  MoveC 5250 to (-74.2, -30.87, -8) mm, rotated rx 180 ry 0 rz 90 deg; joints [72.057, -18.552, 88.853, 0, 19.699, 72.057] to (-74.66, -32.55, -8) mm, rotated rx -180 ry 0 rz 90 deg; joints [71.996, -18.551, 88.847, 0, 19.704, 71.996]
  MoveL 5251 to (-74.66, -70.65, -8) mm, rotated rx 180 ry 0 rz 90 deg; joints [70.74, -18.352, 87.987, 0, 20.365, 70.74]
  MoveC 5252 to (-73.67, -73.03, -8) mm, rotated rx 180 ry 0 rz 90 deg; joints [70.673, -18.323, 87.865, 0, 20.458, 70.673] to (-71.29, -74.01, -8) mm, rotated rx 180 ry 0 rz 90 deg; joints [70.668, -18.28, 87.682, 0, 20.598, 70.668]
  MoveC 5253 to (-53.37, -73.92, -8) mm, rotated rx 180 ry 0 rz 90 deg; joints [70.874, -17.988, 86.471, 0, 21.517, 70.874] to (-35.45, -73.74, -8) mm, rotated rx 180 ry 0 rz 90 deg; joints [71.079, -17.682, 85.244, 0, 22.437, 71.079]
  MoveC 5254 to (-33.46, -73.06, -8) mm, rotated rx 180 ry 0 rz 90 deg; joints [71.123, -17.651, 85.123, 0, 22.528, 71.123] to (-32.27, -71.32, -8) mm, rotated rx 180 ry 0 rz 90 deg; joints [71.192, -17.64, 85.081, 0, 22.559, 71.192]
  MoveC 5255 to (-31.64, -69.07, -8) mm, rotated rx 180 ry 0 rz 90 deg; joints [71.27, -17.643, 85.091, 0, 22.552, 71.27] to (-31.06, -66.81, -8) mm, rotated rx 180 ry 0 rz 90 deg; joints [71.349, -17.646, 85.103, 0, 22.542, 71.349]
  MoveL 5256 to (-30.8, -65.76, -8) mm, rotated rx 180 ry 0 rz 90 deg; joints [71.386, -17.647, 85.11, 0, 22.537, 71.386]
  MoveC 5257 to (-25.24, -44.49, -8) mm, rotated rx -180 ry 0 rz 90 deg; joints [72.129, -17.673, 85.211, 0, 22.462, 72.129] to (-19.72, -23.22, -8) mm, rotated rx -180 ry 0 rz 90 deg; joints [72.873, -17.694, 85.294, 0, 22.401, 72.873]
  MoveC 5258 to (-19.64, -22.75, -8) mm, rotated rx -180 ry 0 rz 90 deg; joints [72.889, -17.695, 85.299, 0, 22.397, 72.889] to (-19.7, -22.27, -8) mm, rotated rx 180 ry 0 rz 90 deg; joints [72.904, -17.699, 85.313, 0, 22.386, 72.904]
  MoveC 5259 to (-20.47, -20.62, -8) mm, rotated rx 180 ry 0 rz 90 deg; joints [72.949, -17.721, 85.402, 0, 22.319, 72.949] to (-21.84, -19.43, -8) mm, rotated rx -180 ry 0 rz 90 deg; joints [72.975, -17.752, 85.523, 0, 22.229, 72.975]
  MoveL 5260 to (-22.21, -19.24, -8) mm, rotated rx -180 ry 0 rz 90 deg; joints [72.977, -17.76, 85.553, 0, 22.206, 72.977]
  MoveC 5261 to (-22.95, -19.01, -8) mm, rotated rx -180 ry 0 rz 90 deg; joints [72.977, -17.774, 85.609, 0, 22.164, 72.977] to (-23.72, -19.03, -8) mm, rotated rx 180 ry 0 rz 90 deg; joints [72.969, -17.787, 85.663, 0, 22.124, 72.969]
  MoveL 5262 to (-32.69, -20.92, -8) mm, rotated rx -180 ry 0 rz 90 deg; joints [72.817, -17.932, 86.244, 0, 21.687, 72.817]
  MoveL 5263 to (-47.78, -24.13, -8) mm, rotated rx 180 ry 0 rz 90 deg; joints [72.558, -18.168, 87.212, 0, 20.956, 72.558]
  MoveL 5264 to (-46.21, -31.51, -8) mm, rotated rx 180 ry 0 rz 90 deg; joints [72.332, -18.103, 86.945, 0, 21.158, 72.332]
  MoveL 5265 to (-46.21, -31.51, -5) mm, rotated rx 180 ry 0 rz 90 deg; joints [72.332, -18.259, 87.047, 0, 21.212, 72.332]
  Establecer velocidad (1000.0 mm/s)
  MoveL 5266 to (-46.21, -31.51, 10) mm, rotated rx 180 ry 0 rz 90 deg; joints [72.332, -19.034, 87.547, 0, 21.486, 72.332]
  Establecer velocidad (66.7 mm/s)
  MoveL 5267 to (15.53, -65.29, 10) mm, rotated rx -180 ry 0 rz 90 deg; joints [71.889, -17.693, 82.447, 0, 25.246, 71.889]
  MoveL 5268 to (15.53, -65.29, -4.75) mm, rotated rx -180 ry 0 rz 90 deg; joints [71.889, -16.947, 81.953, 0, 24.994, 71.889]
  MoveL 5269 to (15.38, -66.79, -5.16) mm, rotated rx 180 ry 0 rz 90 deg; joints [71.84, -16.919, 81.915, 0, 25.005, 71.84]
  MoveL 5270 to (15.6, -68.3, -5.56) mm, rotated rx -180 ry 0 rz 90 deg; joints [71.795, -16.885, 81.85, 0, 25.035, 71.795]
  MoveL 5271 to (16.14, -69.72, -5.97) mm, rotated rx 180 ry 0 rz 90 deg; joints [71.756, -16.844, 81.763, 0, 25.081, 71.756]
  MoveL 5272 to (16.98, -70.99, -6.38) mm, rotated rx -180 ry 0 rz 90 deg; joints [71.725, -16.798, 81.659, 0, 25.14, 71.725]
  MoveL 5273 to (18.08, -72.03, -6.78) mm, rotated rx -180 ry 0 rz 90 deg; joints [71.704, -16.749, 81.54, 0, 25.209, 71.704]
  MoveL 5274 to (19.39, -72.81, -7.19) mm, rotated rx -180 ry 0 rz 90 deg; joints [71.693, -16.697, 81.413, 0, 25.284, 71.693]
  MoveL 5275 to (20.83, -73.28, -7.59) mm, rotated rx 180 ry 0 rz 90 deg; joints [71.693, -16.644, 81.283, 0, 25.361, 71.693]
  MoveL 5276 to (22.34, -73.39, -8) mm, rotated rx -180 ry 0 rz 90 deg; joints [71.705, -16.592, 81.157, 0, 25.435, 71.705]
  MoveC 5277 to (34.58, -73.11, -8) mm, rotated rx 180 ry 0 rz 90 deg; joints [71.839, -16.343, 80.27, 0, 26.073, 71.839] to (46.81, -72.79, -8) mm, rotated rx -180 ry 0 rz 90 deg; joints [71.972, -16.086, 79.374, 0, 26.712, 71.972]
  MoveC 5278 to (49.35, -69.79, -8) mm, rotated rx -180 ry 0 rz 90 deg; joints [72.09, -16.053, 79.258, 0, 26.795, 72.09] to (49.49, -65.86, -8) mm, rotated rx -180 ry 0 rz 90 deg; joints [72.213, -16.077, 79.342, 0, 26.735, 72.213]
  MoveL 5279 to (48.8, -64.98, -8) mm, rotated rx 180 ry 0 rz 90 deg; joints [72.233, -16.098, 79.414, 0, 26.684, 72.233]
  MoveL 5280 to (42.36, -57.33, -8) mm, rotated rx 180 ry 0 rz 90 deg; joints [72.406, -16.286, 80.072, 0, 26.215, 72.406]
  MoveL 5281 to (25.46, -37.43, -8) mm, rotated rx -180 ry 0 rz 90 deg; joints [72.864, -16.761, 81.765, 0, 24.996, 72.864]
  MoveL 5282 to (25.29, -37.24, -8) mm, rotated rx -180 ry 0 rz 90 deg; joints [72.868, -16.765, 81.782, 0, 24.984, 72.868]
  MoveC 5283 to (24.85, -36.79, -8) mm, rotated rx -180 ry 0 rz 90 deg; joints [72.878, -16.777, 81.824, 0, 24.953, 72.878] to (24.37, -36.38, -8) mm, rotated rx 180 ry 0 rz 90 deg; joints [72.886, -16.789, 81.867, 0, 24.921, 72.886]
  MoveL 5284 to (12.74, -27.01, -8) mm, rotated rx -180 ry 0 rz 90 deg; joints [73.07, -17.073, 82.914, 0, 24.159, 73.07]
  MoveL 5285 to (12.32, -26.68, -8) mm, rotated rx -180 ry 0 rz 90 deg; joints [73.077, -17.083, 82.951, 0, 24.132, 73.077]
  MoveC 5286 to (9.55, -26.29, -8) mm, rotated rx -180 ry 0 rz 90 deg; joints [73.062, -17.138, 83.158, 0, 23.98, 73.062] to (7.11, -27.65, -8) mm, rotated rx -180 ry 0 rz 90 deg; joints [72.995, -17.177, 83.303, 0, 23.874, 72.995]
  MoveC 5287 to (6.83, -28.04, -8) mm, rotated rx -180 ry 0 rz 90 deg; joints [72.98, -17.18, 83.314, 0, 23.866, 72.98] to (6.65, -28.48, -8) mm, rotated rx -180 ry 0 rz 90 deg; joints [72.964, -17.181, 83.317, 0, 23.864, 72.964]
  MoveL 5288 to (-4.13, -68.7, -8) mm, rotated rx 180 ry 0 rz 90 deg; joints [71.576, -17.141, 83.169, 0, 23.972, 71.576]
  MoveL 5289 to (-4.25, -69.18, -8) mm, rotated rx 180 ry 0 rz 90 deg; joints [71.56, -17.141, 83.167, 0, 23.974, 71.56]
  MoveC 5290 to (-3.94, -71.7, -8) mm, rotated rx -180 ry 0 rz 90 deg; joints [71.484, -17.119, 83.085, 0, 24.034, 71.484] to (-2.08, -73.44, -8) mm, rotated rx -180 ry 0 rz 90 deg; joints [71.448, -17.072, 82.911, 0, 24.161, 71.448]
  MoveL 5291 to (-1.42, -73.69, -8) mm, rotated rx -180 ry 0 rz 90 deg; joints [71.447, -17.058, 82.858, 0, 24.2, 71.447]
  MoveL 5292 to (-0.47, -73.77, -8) mm, rotated rx 180 ry 0 rz 90 deg; joints [71.455, -17.039, 82.789, 0, 24.25, 71.455]
  MoveC 5293 to (10.93, -73.6, -8) mm, rotated rx -180 ry 0 rz 90 deg; joints [71.58, -16.819, 81.977, 0, 24.842, 71.58] to (22.34, -73.39, -8) mm, rotated rx -180 ry 0 rz 90 deg; joints [71.705, -16.592, 81.157, 0, 25.435, 71.705]
  MoveL 5294 to (22.19, -65.84, -8) mm, rotated rx -180 ry 0 rz 90 deg; joints [71.939, -16.645, 81.348, 0, 25.297, 71.939]
  MoveL 5295 to (22.19, -65.84, -5) mm, rotated rx -180 ry 0 rz 90 deg; joints [71.939, -16.797, 81.45, 0, 25.347, 71.939]
  Establecer velocidad (1000.0 mm/s)
  MoveL 5296 to (22.19, -65.84, 10) mm, rotated rx 180 ry 0 rz 90 deg; joints [71.939, -17.555, 81.953, 0, 25.602, 71.939]
  Establecer velocidad (66.7 mm/s)
  MoveL 5297 to (63.14, -31.68, 10) mm, rotated rx -180 ry 0 rz 90 deg; joints [73.4, -16.913, 79.72, 0, 27.194, 73.4]
  MoveL 5298 to (63.14, -31.68, -4.75) mm, rotated rx -180 ry 0 rz 90 deg; joints [73.4, -16.174, 79.223, 0, 26.951, 73.4]
  MoveL 5299 to (64.65, -31.87, -5.16) mm, rotated rx 180 ry 0 rz 90 deg; joints [73.409, -16.119, 79.092, 0, 27.027, 73.409]
  MoveL 5300 to (66.16, -31.68, -5.56) mm, rotated rx 180 ry 0 rz 90 deg; joints [73.428, -16.067, 78.969, 0, 27.098, 73.428]
  MoveL 5301 to (67.59, -31.17, -5.97) mm, rotated rx 180 ry 0 rz 90 deg; joints [73.457, -16.019, 78.859, 0, 27.16, 73.457]
  MoveL 5302 to (68.87, -30.36, -6.38) mm, rotated rx 180 ry 0 rz 90 deg; joints [73.494, -15.975, 78.766, 0, 27.209, 73.494]
  MoveL 5303 to (69.94, -29.28, -6.78) mm, rotated rx -180 ry 0 rz 90 deg; joints [73.537, -15.938, 78.696, 0, 27.243, 73.537]
  MoveL 5304 to (70.74, -27.99, -7.19) mm, rotated rx 180 ry 0 rz 90 deg; joints [73.584, -15.909, 78.65, 0, 27.259, 73.584]
  MoveL 5305 to (71.24, -26.55, -7.59) mm, rotated rx 180 ry 0 rz 90 deg; joints [73.633, -15.887, 78.63, 0, 27.256, 73.633]
  MoveL 5306 to (71.38, -25.04, -8) mm, rotated rx 180 ry 0 rz 90 deg; joints [73.681, -15.873, 78.639, 0, 27.234, 73.681]
  MoveL 5307 to (71.38, -16.01, -8) mm, rotated rx 180 ry 0 rz 90 deg; joints [73.961, -15.931, 78.837, 0, 27.094, 73.961]
  MoveC 5308 to (69.58, -13.38, -8) mm, rotated rx 180 ry 0 rz 90 deg; joints [74.027, -15.987, 79.03, 0, 26.957, 74.027] to (66.81, -11.79, -8) mm, rotated rx -180 ry 0 rz 90 deg; joints [74.052, -16.057, 79.273, 0, 26.784, 74.052]
  MoveC 5309 to (65.71, -11.6, -8) mm, rotated rx 180 ry 0 rz 90 deg; joints [74.047, -16.082, 79.36, 0, 26.723, 74.047] to (64.59, -11.73, -8) mm, rotated rx -180 ry 0 rz 90 deg; joints [74.034, -16.106, 79.44, 0, 26.665, 74.034]
  MoveL 5310 to (56.12, -23.22, -8) mm, rotated rx 180 ry 0 rz 90 deg; joints [73.599, -16.216, 79.824, 0, 26.392, 73.599]
  MoveL 5311 to (55.62, -23.94, -8) mm, rotated rx -180 ry 0 rz 90 deg; joints [73.572, -16.222, 79.846, 0, 26.376, 73.572]
  MoveC 5312 to (55.02, -26.08, -8) mm, rotated rx -180 ry 0 rz 90 deg; joints [73.5, -16.221, 79.844, 0, 26.378, 73.5] to (55.87, -28.13, -8) mm, rotated rx 180 ry 0 rz 90 deg; joints [73.444, -16.19, 79.735, 0, 26.456, 73.444]
  MoveL 5313 to (64.98, -38.32, -8) mm, rotated rx -180 ry 0 rz 90 deg; joints [73.212, -15.927, 78.824, 0, 27.103, 73.212]
  MoveC 5314 to (66.47, -38.38, -8) mm, rotated rx 180 ry 0 rz 90 deg; joints [73.224, -15.894, 78.711, 0, 27.183, 73.224] to (67.89, -37.93, -8) mm, rotated rx -180 ry 0 rz 90 deg; joints [73.251, -15.866, 78.614, 0, 27.251, 73.251]
  MoveL 5315 to (68.22, -37.76, -8) mm, rotated rx 180 ry 0 rz 90 deg; joints [73.259, -15.859, 78.593, 0, 27.266, 73.259]
  MoveC 5316 to (70.16, -36.22, -8) mm, rotated rx -180 ry 0 rz 90 deg; joints [73.325, -15.827, 78.482, 0, 27.345, 73.325] to (71.38, -34.07, -8) mm, rotated rx -180 ry 0 rz 90 deg; joints [73.402, -15.814, 78.437, 0, 27.376, 73.402]
  MoveL 5317 to (71.38, -25.04, -8) mm, rotated rx 180 ry 0 rz 90 deg; joints [73.681, -15.873, 78.639, 0, 27.234, 73.681]
  MoveL 5318 to (63.83, -25.04, -8) mm, rotated rx 180 ry 0 rz 90 deg; joints [73.613, -16.038, 79.208, 0, 26.831, 73.613]
  MoveL 5319 to (63.83, -25.48, -8) mm, rotated rx -180 ry 0 rz 90 deg; joints [73.599, -16.036, 79.198, 0, 26.838, 73.599]
  MoveL 5320 to (63.83, -25.48, -5) mm, rotated rx 180 ry 0 rz 90 deg; joints [73.599, -16.186, 79.301, 0, 26.886, 73.599]
  Establecer velocidad (1000.0 mm/s)
  MoveL 5321 to (63.83, -25.48, 10) mm, rotated rx -180 ry 0 rz 90 deg; joints [73.599, -16.939, 79.806, 0, 27.133, 73.599]
  Establecer velocidad (66.7 mm/s)
  MoveL 5322 to (31.82, 9.28, 10) mm, rotated rx -180 ry 0 rz 90 deg; joints [74.404, -17.82, 82.904, 0, 24.916, 74.404]
  MoveL 5323 to (31.82, 9.28, -4.75) mm, rotated rx 180 ry 0 rz 90 deg; joints [74.404, -17.072, 82.41, 0, 24.662, 74.404]
  MoveL 5324 to (32.94, 8.26, -5.16) mm, rotated rx 180 ry 0 rz 90 deg; joints [74.381, -17.024, 82.294, 0, 24.729, 74.381]
  MoveL 5325 to (34.28, 7.54, -5.56) mm, rotated rx 180 ry 0 rz 90 deg; joints [74.37, -16.972, 82.168, 0, 24.804, 74.37]
  MoveL 5326 to (35.74, 7.13, -5.97) mm, rotated rx -180 ry 0 rz 90 deg; joints [74.37, -16.92, 82.039, 0, 24.881, 74.37]
  MoveL 5327 to (37.26, 7.06, -6.38) mm, rotated rx 180 ry 0 rz 90 deg; joints [74.382, -16.869, 81.913, 0, 24.955, 74.382]
  MoveL 5328 to (38.76, 7.32, -6.78) mm, rotated rx 180 ry 0 rz 90 deg; joints [74.403, -16.819, 81.795, 0, 25.024, 74.403]
  MoveL 5329 to (40.15, 7.91, -7.19) mm, rotated rx 180 ry 0 rz 90 deg; joints [74.434, -16.774, 81.691, 0, 25.083, 74.434]
  MoveL 5330 to (41.39, 8.8, -7.59) mm, rotated rx 180 ry 0 rz 90 deg; joints [74.473, -16.733, 81.605, 0, 25.129, 74.473]
  MoveL 5331 to (42.37, 9.95, -8) mm, rotated rx 180 ry 0 rz 90 deg; joints [74.519, -16.699, 81.542, 0, 25.157, 74.519]
  MoveL 5332 to (51.07, 22.27, -8) mm, rotated rx 180 ry 0 rz 90 deg; joints [74.985, -16.59, 81.149, 0, 25.441, 74.985]
  MoveC 5333 to (50.81, 26.19, -8) mm, rotated rx 180 ry 0 rz 90 deg; joints [75.107, -16.617, 81.245, 0, 25.371, 75.107] to (48.1, 29.04, -8) mm, rotated rx 180 ry 0 rz 90 deg; joints [75.175, -16.688, 81.501, 0, 25.187, 75.175]
  MoveC 5334 to (29.5, 28.81, -8) mm, rotated rx -180 ry 0 rz 90 deg; joints [75.009, -17.057, 82.856, 0, 24.201, 75.009] to (10.9, 28.45, -8) mm, rotated rx 180 ry 0 rz 90 deg; joints [74.836, -17.41, 84.188, 0, 23.222, 74.836]
  MoveC 5335 to (8.09, 27.12, -8) mm, rotated rx 180 ry 0 rz 90 deg; joints [74.768, -17.455, 84.362, 0, 23.093, 74.768] to (7.1, 24.17, -8) mm, rotated rx 180 ry 0 rz 90 deg; joints [74.663, -17.459, 84.375, 0, 23.084, 74.663]
  MoveC 5336 to (7.15, 23.93, -8) mm, rotated rx 180 ry 0 rz 90 deg; joints [74.656, -17.457, 84.367, 0, 23.089, 74.656] to (7.21, 23.7, -8) mm, rotated rx -180 ry 0 rz 90 deg; joints [74.649, -17.454, 84.358, 0, 23.096, 74.649]
  MoveL 5337 to (11.88, 10.9, -8) mm, rotated rx -180 ry 0 rz 90 deg; joints [74.277, -17.301, 83.771, 0, 23.53, 74.277]
  MoveL 5338 to (12.28, 9.83, -8) mm, rotated rx -180 ry 0 rz 90 deg; joints [74.246, -17.288, 83.721, 0, 23.567, 74.246]
  MoveC 5339 to (12.77, 8.93, -8) mm, rotated rx 180 ry 0 rz 90 deg; joints [74.221, -17.274, 83.668, 0, 23.606, 74.221] to (13.49, 8.19, -8) mm, rotated rx -180 ry 0 rz 90 deg; joints [74.204, -17.256, 83.601, 0, 23.655, 74.204]
  MoveL 5340 to (27.96, -2.86, -8) mm, rotated rx -180 ry 0 rz 90 deg; joints [73.982, -16.915, 82.331, 0, 24.585, 73.982]
  MoveL 5341 to (28.9, -3.52, -8) mm, rotated rx 180 ry 0 rz 90 deg; joints [73.97, -16.893, 82.248, 0, 24.645, 73.97]
  MoveC 5342 to (31.47, -3.69, -8) mm, rotated rx -180 ry 0 rz 90 deg; joints [73.988, -16.841, 82.058, 0, 24.783, 73.988] to (33.68, -2.37, -8) mm, rotated rx -180 ry 0 rz 90 deg; joints [74.05, -16.804, 81.924, 0, 24.88, 74.05]
  MoveL 5343 to (42.37, 9.95, -8) mm, rotated rx 180 ry 0 rz 90 deg; joints [74.519, -16.699, 81.542, 0, 25.157, 74.519]
  MoveL 5344 to (36.21, 14.3, -8) mm, rotated rx -180 ry 0 rz 90 deg; joints [74.603, -16.847, 82.081, 0, 24.766, 74.603]
  MoveL 5345 to (36.21, 14.3, -5) mm, rotated rx 180 ry 0 rz 90 deg; joints [74.603, -17, 82.183, 0, 24.816, 74.603]
  Establecer velocidad (1000.0 mm/s)
  MoveL 5346 to (36.21, 14.3, 10) mm, rotated rx 180 ry 0 rz 90 deg; joints [74.603, -17.76, 82.686, 0, 25.074, 74.603]
  Establecer velocidad (66.7 mm/s)
  MoveL 5347 to (28.17, 64.78, 10) mm, rotated rx 180 ry 0 rz 90 deg; joints [76.16, -18.179, 84.225, 0, 23.954, 76.16]
  MoveL 5348 to (28.17, 64.78, -4.75) mm, rotated rx 180 ry 0 rz 90 deg; joints [76.16, -17.427, 83.732, 0, 23.695, 76.16]
  MoveL 5349 to (28.39, 66.28, -5.16) mm, rotated rx -180 ry 0 rz 90 deg; joints [76.21, -17.41, 83.729, 0, 23.68, 76.21]
  MoveL 5350 to (28.24, 67.79, -5.56) mm, rotated rx 180 ry 0 rz 90 deg; joints [76.258, -17.399, 83.753, 0, 23.645, 76.258]
  MoveL 5351 to (27.76, 69.23, -5.97) mm, rotated rx 180 ry 0 rz 90 deg; joints [76.302, -17.394, 83.8, 0, 23.594, 76.302]
  MoveL 5352 to (26.97, 70.53, -6.38) mm, rotated rx 180 ry 0 rz 90 deg; joints [76.338, -17.394, 83.865, 0, 23.529, 76.338]
  MoveL 5353 to (25.91, 71.63, -6.78) mm, rotated rx -180 ry 0 rz 90 deg; joints [76.365, -17.398, 83.947, 0, 23.451, 76.365]
  MoveL 5354 to (24.64, 72.46, -7.19) mm, rotated rx 180 ry 0 rz 90 deg; joints [76.382, -17.405, 84.039, 0, 23.366, 76.382]
  MoveL 5355 to (23.22, 72.99, -7.59) mm, rotated rx -180 ry 0 rz 90 deg; joints [76.388, -17.414, 84.137, 0, 23.277, 76.388]
  MoveL 5356 to (21.71, 73.16, -8) mm, rotated rx -180 ry 0 rz 90 deg; joints [76.382, -17.422, 84.235, 0, 23.187, 76.382]
  MoveL 5357 to (16.58, 73.28, -8) mm, rotated rx -180 ry 0 rz 90 deg; joints [76.345, -17.518, 84.605, 0, 22.913, 76.345]
  MoveL 5358 to (-23.22, 73.93, -8) mm, rotated rx 180 ry 0 rz 90 deg; joints [76.043, -18.217, 87.419, 0, 20.798, 76.043]
  MoveL 5359 to (-24.65, 73.95, -8) mm, rotated rx 180 ry 0 rz 90 deg; joints [76.031, -18.241, 87.519, 0, 20.722, 76.031]
  MoveC 5360 to (-27.16, 70.81, -8) mm, rotated rx -180 ry 0 rz 90 deg; joints [75.905, -18.269, 87.638, 0, 20.632, 75.905] to (-26.78, 66.82, -8) mm, rotated rx 180 ry 0 rz 90 deg; joints [75.774, -18.247, 87.542, 0, 20.705, 75.774]
  MoveL 5361 to (-9, 55.49, -8) mm, rotated rx 180 ry 0 rz 90 deg; joints [75.549, -17.897, 86.102, 0, 21.795, 75.549]
  MoveL 5362 to (-8.91, 55.44, -8) mm, rotated rx -180 ry 0 rz 90 deg; joints [75.548, -17.895, 86.094, 0, 21.801, 75.548]
  MoveL 5363 to (-8.41, 55.2, -8) mm, rotated rx -180 ry 0 rz 90 deg; joints [75.544, -17.885, 86.055, 0, 21.83, 75.544]
  MoveL 5364 to (-8.28, 55.16, -8) mm, rotated rx -180 ry 0 rz 90 deg; joints [75.544, -17.883, 86.046, 0, 21.837, 75.544]
  MoveC 5365 to (-7.7, 55.1, -8) mm, rotated rx 180 ry 0 rz 90 deg; joints [75.547, -17.872, 86.004, 0, 21.869, 75.547] to (-7.11, 55.11, -8) mm, rotated rx 180 ry 0 rz 90 deg; joints [75.552, -17.862, 85.962, 0, 21.9, 75.552]
  MoveC 5366 to (9.95, 56.35, -8) mm, rotated rx 180 ry 0 rz 90 deg; joints [75.737, -17.562, 84.778, 0, 22.785, 75.737] to (27.01, 57.72, -8) mm, rotated rx 180 ry 0 rz 90 deg; joints [75.922, -17.25, 83.579, 0, 23.671, 75.922]
  MoveC 5367 to (45.69, 59.55, -8) mm, rotated rx -180 ry 0 rz 90 deg; joints [76.131, -16.894, 82.252, 0, 24.642, 76.131] to (64.31, 62.01, -8) mm, rotated rx 180 ry 0 rz 90 deg; joints [76.355, -16.526, 80.92, 0, 25.606, 76.355]
  MoveC 5368 to (66.34, 62.34, -8) mm, rotated rx 180 ry 0 rz 90 deg; joints [76.381, -16.485, 80.774, 0, 25.711, 76.381] to (68.36, 62.74, -8) mm, rotated rx 180 ry 0 rz 90 deg; joints [76.41, -16.445, 80.631, 0, 25.814, 76.41]
  MoveC 5369 to (69.69, 63.56, -8) mm, rotated rx -180 ry 0 rz 90 deg; joints [76.446, -16.421, 80.545, 0, 25.875, 76.446] to (70.22, 65.04, -8) mm, rotated rx 180 ry 0 rz 90 deg; joints [76.497, -16.417, 80.533, 0, 25.884, 76.497]
  MoveL 5370 to (70.22, 68.58, -8) mm, rotated rx -180 ry 0 rz 90 deg; joints [76.61, -16.435, 80.596, 0, 25.839, 76.61]
  MoveC 5371 to (69.59, 70.2, -8) mm, rotated rx 180 ry 0 rz 90 deg; joints [76.656, -16.456, 80.672, 0, 25.784, 76.656] to (68.02, 70.96, -8) mm, rotated rx 180 ry 0 rz 90 deg; joints [76.669, -16.493, 80.803, 0, 25.69, 76.669]
  MoveC 5372 to (46.54, 72.32, -8) mm, rotated rx 180 ry 0 rz 90 deg; joints [76.548, -16.939, 82.418, 0, 24.521, 76.548] to (25.02, 73.09, -8) mm, rotated rx -180 ry 0 rz 90 deg; joints [76.406, -17.36, 83.995, 0, 23.364, 76.406]
  MoveL 5373 to (21.71, 73.16, -8) mm, rotated rx -180 ry 0 rz 90 deg; joints [76.382, -17.422, 84.235, 0, 23.187, 76.382]
  MoveL 5374 to (21.54, 65.62, -8) mm, rotated rx -180 ry 0 rz 90 deg; joints [76.134, -17.391, 84.114, 0, 23.276, 76.134]
  MoveL 5375 to (21.54, 65.62, -5) mm, rotated rx -180 ry 0 rz 90 deg; joints [76.134, -17.544, 84.216, 0, 23.328, 76.134]
  Establecer velocidad (1000.0 mm/s)
  MoveL 5376 to (21.54, 65.62, 10) mm, rotated rx -180 ry 0 rz 90 deg; joints [76.134, -18.31, 84.717, 0, 23.593, 76.134]
  Establecer velocidad (66.7 mm/s)
  MoveL 5377 to (28.17, 64.55, 10) mm, rotated rx 180 ry 0 rz 90 deg; joints [76.152, -18.178, 84.221, 0, 23.957, 76.152]
  MoveL 5378 to (28.17, 64.55, -5) mm, rotated rx -180 ry 0 rz 90 deg; joints [76.152, -17.413, 83.72, 0, 23.694, 76.152]
  MoveL 5379 to (28.38, 66.05, -5.41) mm, rotated rx -180 ry 0 rz 90 deg; joints [76.203, -17.396, 83.717, 0, 23.679, 76.203]
  MoveL 5380 to (28.23, 67.56, -5.81) mm, rotated rx 180 ry 0 rz 90 deg; joints [76.251, -17.385, 83.741, 0, 23.644, 76.251]
  MoveL 5381 to (27.75, 69, -6.22) mm, rotated rx 180 ry 0 rz 90 deg; joints [76.294, -17.38, 83.787, 0, 23.593, 76.294]
  MoveL 5382 to (26.96, 70.3, -6.62) mm, rotated rx 180 ry 0 rz 90 deg; joints [76.33, -17.38, 83.853, 0, 23.527, 76.33]
  MoveL 5383 to (25.91, 71.39, -7.03) mm, rotated rx -180 ry 0 rz 90 deg; joints [76.357, -17.385, 83.935, 0, 23.45, 76.357]
  MoveL 5384 to (24.64, 72.23, -7.44) mm, rotated rx -180 ry 0 rz 90 deg; joints [76.374, -17.392, 84.027, 0, 23.365, 76.374]
  MoveL 5385 to (23.21, 72.76, -7.84) mm, rotated rx -180 ry 0 rz 90 deg; joints [76.38, -17.4, 84.125, 0, 23.275, 76.38]
  MoveL 5386 to (21.71, 72.93, -8.25) mm, rotated rx -180 ry 0 rz 90 deg; joints [76.374, -17.408, 84.223, 0, 23.186, 76.374]
  MoveC 5387 to (-1.16, 73.38, -8.25) mm, rotated rx -180 ry 0 rz 90 deg; joints [76.206, -17.825, 85.858, 0, 21.967, 76.206] to (-24.02, 73.75, -8.25) mm, rotated rx -180 ry 0 rz 90 deg; joints [76.03, -18.217, 87.463, 0, 20.754, 76.03]
  MoveC 5388 to (-26.51, 70.65, -8.25) mm, rotated rx -180 ry 0 rz 90 deg; joints [75.905, -18.245, 87.582, 0, 20.663, 75.905] to (-26.15, 66.69, -8.25) mm, rotated rx 180 ry 0 rz 90 deg; joints [75.776, -18.223, 87.487, 0, 20.735, 75.776]
  MoveL 5389 to (-24.87, 65.86, -8.25) mm, rotated rx 180 ry 0 rz 90 deg; joints [75.759, -18.198, 87.384, 0, 20.814, 75.759]
  MoveL 5390 to (-10.9, 56.96, -8.25) mm, rotated rx 180 ry 0 rz 90 deg; joints [75.581, -17.923, 86.253, 0, 21.67, 75.581]
  MoveL 5391 to (-9, 55.75, -8.25) mm, rotated rx 180 ry 0 rz 90 deg; joints [75.557, -17.885, 86.098, 0, 21.787, 75.557]
  MoveL 5392 to (-8.24, 55.35, -8.25) mm, rotated rx 180 ry 0 rz 90 deg; joints [75.551, -17.87, 86.037, 0, 21.833, 75.551]
  MoveL 5393 to (-8.05, 55.29, -8.25) mm, rotated rx 180 ry 0 rz 90 deg; joints [75.55, -17.866, 86.023, 0, 21.843, 75.55]
  MoveC 5394 to (-7.63, 55.26, -8.25) mm, rotated rx -180 ry 0 rz 90 deg; joints [75.553, -17.859, 85.993, 0, 21.866, 75.553] to (-7.2, 55.27, -8.25) mm, rotated rx 180 ry 0 rz 90 deg; joints [75.557, -17.851, 85.963, 0, 21.889, 75.557]
  MoveC 5395 to (9.44, 56.48, -8.25) mm, rotated rx 180 ry 0 rz 90 deg; joints [75.736, -17.56, 84.808, 0, 22.752, 75.736] to (26.06, 57.83, -8.25) mm, rotated rx 180 ry 0 rz 90 deg; joints [75.917, -17.256, 83.641, 0, 23.615, 75.917]
  MoveL 5396 to (32.37, 58.4, -8.25) mm, rotated rx 180 ry 0 rz 90 deg; joints [75.987, -17.138, 83.194, 0, 23.943, 75.987]
  MoveC 5397 to (50.11, 60.34, -8.25) mm, rotated rx 180 ry 0 rz 90 deg; joints [76.191, -16.797, 81.933, 0, 24.863, 76.191] to (67.76, 62.94, -8.25) mm, rotated rx 180 ry 0 rz 90 deg; joints [76.412, -16.446, 80.671, 0, 25.775, 76.412]
  MoveL 5398 to (68.22, 63.07, -8.25) mm, rotated rx -180 ry 0 rz 90 deg; joints [76.419, -16.437, 80.638, 0, 25.799, 76.419]
  MoveC 5399 to (69.42, 63.87, -8.25) mm, rotated rx 180 ry 0 rz 90 deg; joints [76.454, -16.416, 80.563, 0, 25.852, 76.454] to (69.88, 65.22, -8.25) mm, rotated rx 180 ry 0 rz 90 deg; joints [76.5, -16.413, 80.553, 0, 25.86, 76.5]
  MoveL 5400 to (69.89, 68.7, -8.25) mm, rotated rx 180 ry 0 rz 90 deg; joints [76.611, -16.43, 80.614, 0, 25.816, 76.611]
  MoveC 5401 to (69.18, 70.06, -8.25) mm, rotated rx 180 ry 0 rz 90 deg; joints [76.649, -16.452, 80.692, 0, 25.76, 76.649] to (67.76, 70.63, -8.25) mm, rotated rx -180 ry 0 rz 90 deg; joints [76.656, -16.485, 80.808, 0, 25.676, 76.656]
  MoveC 5402 to (45.03, 72.12, -8.25) mm, rotated rx 180 ry 0 rz 90 deg; joints [76.53, -16.955, 82.516, 0, 24.439, 76.53] to (22.27, 72.92, -8.25) mm, rotated rx -180 ry 0 rz 90 deg; joints [76.378, -17.398, 84.182, 0, 23.216, 76.378]
  MoveC 5403 to (21.99, 72.92, -8.25) mm, rotated rx -180 ry 0 rz 90 deg; joints [76.376, -17.403, 84.202, 0, 23.201, 76.376] to (21.71, 72.93, -8.25) mm, rotated rx -180 ry 0 rz 90 deg; joints [76.374, -17.408, 84.223, 0, 23.186, 76.374]
  MoveL 5404 to (21.54, 65.38, -8.25) mm, rotated rx -180 ry 0 rz 90 deg; joints [76.126, -17.377, 84.102, 0, 23.275, 76.126]
  MoveL 5405 to (21.54, 65.38, -5.25) mm, rotated rx 180 ry 0 rz 90 deg; joints [76.126, -17.53, 84.204, 0, 23.327, 76.126]
  Establecer velocidad (1000.0 mm/s)
  MoveL 5406 to (21.54, 65.38, 10) mm, rotated rx 180 ry 0 rz 90 deg; joints [76.126, -18.309, 84.713, 0, 23.596, 76.126]
  Establecer velocidad (66.7 mm/s)
  MoveL 5407 to (36.05, 20.42, 10) mm, rotated rx -180 ry 0 rz 90 deg; joints [74.797, -17.797, 82.82, 0, 24.977, 74.797]
  MoveL 5408 to (36.05, 20.42, -5) mm, rotated rx 180 ry 0 rz 90 deg; joints [74.797, -17.036, 82.317, 0, 24.719, 74.797]
  MoveL 5409 to (36.21, 21.93, -5.41) mm, rotated rx 180 ry 0 rz 90 deg; joints [74.847, -17.021, 82.322, 0, 24.699, 74.847]
  MoveL 5410 to (36, 23.44, -5.81) mm, rotated rx 180 ry 0 rz 90 deg; joints [74.893, -17.012, 82.353, 0, 24.66, 74.893]
  MoveL 5411 to (35.47, 24.86, -6.22) mm, rotated rx 180 ry 0 rz 90 deg; joints [74.934, -17.01, 82.406, 0, 24.604, 74.934]
  MoveL 5412 to (34.64, 26.13, -6.62) mm, rotated rx 180 ry 0 rz 90 deg; joints [74.967, -17.013, 82.478, 0, 24.535, 74.967]
  MoveL 5413 to (33.54, 27.19, -7.03) mm, rotated rx -180 ry 0 rz 90 deg; joints [74.992, -17.019, 82.564, 0, 24.455, 74.992]
  MoveL 5414 to (32.24, 27.97, -7.44) mm, rotated rx -180 ry 0 rz 90 deg; joints [75.006, -17.028, 82.66, 0, 24.368, 75.006]
  MoveL 5415 to (30.8, 28.45, -7.84) mm, rotated rx -180 ry 0 rz 90 deg; joints [75.008, -17.038, 82.76, 0, 24.278, 75.008]
  MoveL 5416 to (29.28, 28.56, -8.25) mm, rotated rx 180 ry 0 rz 90 deg; joints [74.999, -17.048, 82.859, 0, 24.189, 74.999]
  MoveC 5417 to (20.09, 28.41, -8.25) mm, rotated rx -180 ry 0 rz 90 deg; joints [74.915, -17.224, 83.52, 0, 23.704, 74.915] to (10.9, 28.22, -8.25) mm, rotated rx 180 ry 0 rz 90 deg; joints [74.828, -17.396, 84.175, 0, 23.221, 74.828]
  MoveC 5418 to (8.21, 26.7, -8.25) mm, rotated rx -180 ry 0 rz 90 deg; joints [74.755, -17.438, 84.337, 0, 23.101, 74.755] to (7.48, 23.69, -8.25) mm, rotated rx -180 ry 0 rz 90 deg; joints [74.651, -17.437, 84.331, 0, 23.106, 74.651]
  MoveL 5419 to (7.64, 23.22, -8.25) mm, rotated rx -180 ry 0 rz 90 deg; joints [74.637, -17.431, 84.31, 0, 23.121, 74.637]
  MoveL 5420 to (12.13, 10.9, -8.25) mm, rotated rx -180 ry 0 rz 90 deg; joints [74.279, -17.283, 83.744, 0, 23.539, 74.279]
  MoveL 5421 to (12.5, 9.9, -8.25) mm, rotated rx 180 ry 0 rz 90 deg; joints [74.25, -17.271, 83.698, 0, 23.573, 74.25]
  MoveC 5422 to (12.93, 9.1, -8.25) mm, rotated rx 180 ry 0 rz 90 deg; joints [74.228, -17.259, 83.651, 0, 23.608, 74.228] to (13.56, 8.45, -8.25) mm, rotated rx -180 ry 0 rz 90 deg; joints [74.213, -17.243, 83.593, 0, 23.651, 74.213]
  MoveL 5423 to (14.06, 8.05, -8.25) mm, rotated rx 180 ry 0 rz 90 deg; joints [74.205, -17.232, 83.549, 0, 23.683, 74.205]
  MoveL 5424 to (27.96, -2.54, -8.25) mm, rotated rx -180 ry 0 rz 90 deg; joints [73.992, -16.905, 82.329, 0, 24.576, 73.992]
  MoveL 5425 to (28.9, -3.2, -8.25) mm, rotated rx 180 ry 0 rz 90 deg; joints [73.98, -16.882, 82.246, 0, 24.636, 73.98]
  MoveC 5426 to (31.65, -3.31, -8.25) mm, rotated rx -180 ry 0 rz 90 deg; joints [74.002, -16.827, 82.044, 0, 24.783, 74.002] to (33.88, -1.7, -8.25) mm, rotated rx 180 ry 0 rz 90 deg; joints [74.073, -16.792, 81.915, 0, 24.876, 74.073]
  MoveL 5427 to (49.44, 20.37, -8.25) mm, rotated rx 180 ry 0 rz 90 deg; joints [74.911, -16.6, 81.223, 0, 25.377, 74.911]
  MoveL 5428 to (50.44, 21.83, -8.25) mm, rotated rx 180 ry 0 rz 90 deg; joints [74.965, -16.588, 81.178, 0, 25.41, 74.965]
  MoveC 5429 to (50.85, 23.18, -8.25) mm, rotated rx -180 ry 0 rz 90 deg; joints [75.012, -16.587, 81.175, 0, 25.412, 75.012] to (50.7, 24.58, -8.25) mm, rotated rx 180 ry 0 rz 90 deg; joints [75.055, -16.598, 81.214, 0, 25.384, 75.055]
  MoveC 5430 to (49.7, 27.05, -8.25) mm, rotated rx 180 ry 0 rz 90 deg; joints [75.125, -16.632, 81.336, 0, 25.296, 75.125] to (47.67, 28.77, -8.25) mm, rotated rx 180 ry 0 rz 90 deg; joints [75.162, -16.682, 81.519, 0, 25.164, 75.162]
  MoveC 5431 to (38.48, 28.68, -8.25) mm, rotated rx 180 ry 0 rz 90 deg; joints [75.082, -16.867, 82.192, 0, 24.676, 75.082] to (29.28, 28.56, -8.25) mm, rotated rx 180 ry 0 rz 90 deg; joints [74.999, -17.048, 82.859, 0, 24.189, 74.999]
  MoveL 5432 to (29.4, 21.02, -8.25) mm, rotated rx -180 ry 0 rz 90 deg; joints [74.758, -17.006, 82.702, 0, 24.303, 74.758]
  MoveL 5433 to (29.4, 21.02, -5.25) mm, rotated rx 180 ry 0 rz 90 deg; joints [74.758, -17.158, 82.804, 0, 24.354, 74.758]
  Establecer velocidad (1000.0 mm/s)
  MoveL 5434 to (29.4, 21.02, 10) mm, rotated rx 180 ry 0 rz 90 deg; joints [74.758, -17.933, 83.315, 0, 24.618, 74.758]
  Establecer velocidad (66.7 mm/s)
  MoveL 5435 to (62.87, -31.77, 10) mm, rotated rx -180 ry 0 rz 90 deg; joints [73.395, -16.919, 79.738, 0, 27.181, 73.395]
  MoveL 5436 to (62.87, -31.77, -5) mm, rotated rx 180 ry 0 rz 90 deg; joints [73.395, -16.167, 79.233, 0, 26.934, 73.395]
  MoveL 5437 to (64.38, -31.95, -5.41) mm, rotated rx -180 ry 0 rz 90 deg; joints [73.403, -16.112, 79.102, 0, 27.01, 73.403]
  MoveL 5438 to (65.89, -31.77, -5.81) mm, rotated rx 180 ry 0 rz 90 deg; joints [73.423, -16.06, 78.979, 0, 27.081, 73.423]
  MoveL 5439 to (67.32, -31.25, -6.22) mm, rotated rx 180 ry 0 rz 90 deg; joints [73.452, -16.012, 78.869, 0, 27.143, 73.452]
  MoveL 5440 to (68.6, -30.44, -6.62) mm, rotated rx 180 ry 0 rz 90 deg; joints [73.489, -15.968, 78.776, 0, 27.192, 73.489]
  MoveL 5441 to (69.67, -29.36, -7.03) mm, rotated rx 180 ry 0 rz 90 deg; joints [73.532, -15.931, 78.706, 0, 27.225, 73.532]
  MoveL 5442 to (70.47, -28.07, -7.44) mm, rotated rx 180 ry 0 rz 90 deg; joints [73.579, -15.902, 78.66, 0, 27.242, 73.579]
  MoveL 5443 to (70.97, -26.64, -7.84) mm, rotated rx 180 ry 0 rz 90 deg; joints [73.628, -15.879, 78.64, 0, 27.239, 73.628]
  MoveL 5444 to (71.11, -25.13, -8.25) mm, rotated rx 180 ry 0 rz 90 deg; joints [73.676, -15.866, 78.649, 0, 27.217, 73.676]
  MoveL 5445 to (71.11, -16.72, -8.25) mm, rotated rx -180 ry 0 rz 90 deg; joints [73.937, -15.92, 78.833, 0, 27.086, 73.937]
  MoveC 5446 to (69.41, -14.18, -8.25) mm, rotated rx -180 ry 0 rz 90 deg; joints [74, -15.973, 79.017, 0, 26.956, 74] to (66.81, -12.57, -8.25) mm, rotated rx 180 ry 0 rz 90 deg; joints [74.027, -16.04, 79.247, 0, 26.792, 74.027]
  MoveC 5447 to (65.62, -12.33, -8.25) mm, rotated rx 180 ry 0 rz 90 deg; joints [74.024, -16.067, 79.342, 0, 26.725, 74.024] to (64.42, -12.43, -8.25) mm, rotated rx 180 ry 0 rz 90 deg; joints [74.01, -16.092, 79.43, 0, 26.663, 74.01]
  MoveL 5448 to (56.39, -23.31, -8.25) mm, rotated rx 180 ry 0 rz 90 deg; joints [73.598, -16.197, 79.794, 0, 26.403, 73.598]
  MoveL 5449 to (55.95, -23.93, -8.25) mm, rotated rx 180 ry 0 rz 90 deg; joints [73.575, -16.202, 79.813, 0, 26.39, 73.575]
  MoveC 5450 to (55.35, -26.06, -8.25) mm, rotated rx -180 ry 0 rz 90 deg; joints [73.503, -16.202, 79.811, 0, 26.391, 73.503] to (56.2, -28.11, -8.25) mm, rotated rx -180 ry 0 rz 90 deg; joints [73.447, -16.171, 79.702, 0, 26.469, 73.447]
  MoveL 5451 to (64.81, -37.7, -8.25) mm, rotated rx 180 ry 0 rz 90 deg; joints [73.229, -15.922, 78.843, 0, 27.08, 73.229]
  MoveC 5452 to (67.03, -37.57, -8.25) mm, rotated rx 180 ry 0 rz 90 deg; joints [73.254, -15.874, 78.678, 0, 27.196, 73.254] to (68.98, -36.48, -8.25) mm, rotated rx 180 ry 0 rz 90 deg; joints [73.306, -15.839, 78.556, 0, 27.282, 73.306]
  MoveL 5453 to (69.36, -36.13, -8.25) mm, rotated rx 180 ry 0 rz 90 deg; joints [73.32, -15.832, 78.535, 0, 27.297, 73.32]
  MoveC 5454 to (70.39, -34.93, -8.25) mm, rotated rx -180 ry 0 rz 90 deg; joints [73.367, -15.818, 78.484, 0, 27.333, 73.367] to (71.1, -33.53, -8.25) mm, rotated rx 180 ry 0 rz 90 deg; joints [73.417, -15.811, 78.462, 0, 27.349, 73.417]
  MoveL 5455 to (71.11, -32.69, -8.25) mm, rotated rx 180 ry 0 rz 90 deg; joints [73.442, -15.816, 78.48, 0, 27.336, 73.442]
  MoveL 5456 to (71.11, -25.13, -8.25) mm, rotated rx 180 ry 0 rz 90 deg; joints [73.676, -15.866, 78.649, 0, 27.217, 73.676]
  MoveL 5457 to (63.56, -25.13, -8.25) mm, rotated rx 180 ry 0 rz 90 deg; joints [73.608, -16.031, 79.218, 0, 26.813, 73.608]
  MoveL 5458 to (63.56, -25.13, -5.25) mm, rotated rx -180 ry 0 rz 90 deg; joints [73.608, -16.182, 79.32, 0, 26.862, 73.608]
  Establecer velocidad (1000.0 mm/s)
  MoveL 5459 to (63.56, -25.13, 10) mm, rotated rx -180 ry 0 rz 90 deg; joints [73.608, -16.947, 79.834, 0, 27.113, 73.608]
  Establecer velocidad (66.7 mm/s)
  MoveL 5460 to (16.2, -65.05, 10) mm, rotated rx -180 ry 0 rz 90 deg; joints [71.903, -17.682, 82.405, 0, 25.276, 71.903]
  MoveL 5461 to (16.2, -65.05, -5) mm, rotated rx -180 ry 0 rz 90 deg; joints [71.903, -16.922, 81.903, 0, 25.02, 71.903]
  MoveL 5462 to (16.05, -66.56, -5.41) mm, rotated rx -180 ry 0 rz 90 deg; joints [71.854, -16.895, 81.864, 0, 25.031, 71.854]
  MoveL 5463 to (16.26, -68.06, -5.81) mm, rotated rx 180 ry 0 rz 90 deg; joints [71.809, -16.86, 81.799, 0, 25.061, 71.809]
  MoveL 5464 to (16.8, -69.48, -6.22) mm, rotated rx -180 ry 0 rz 90 deg; joints [71.77, -16.82, 81.712, 0, 25.107, 71.77]
  MoveL 5465 to (17.65, -70.75, -6.62) mm, rotated rx -180 ry 0 rz 90 deg; joints [71.739, -16.774, 81.607, 0, 25.167, 71.739]
  MoveL 5466 to (18.75, -71.79, -7.03) mm, rotated rx -180 ry 0 rz 90 deg; joints [71.718, -16.724, 81.489, 0, 25.236, 71.718]
  MoveL 5467 to (20.06, -72.57, -7.44) mm, rotated rx 180 ry 0 rz 90 deg; joints [71.707, -16.672, 81.362, 0, 25.311, 71.707]
  MoveL 5468 to (21.5, -73.04, -7.84) mm, rotated rx -180 ry 0 rz 90 deg; joints [71.708, -16.62, 81.232, 0, 25.388, 71.708]
  MoveL 5469 to (23.02, -73.14, -8.25) mm, rotated rx 180 ry 0 rz 90 deg; joints [71.72, -16.568, 81.105, 0, 25.462, 71.72]
  MoveC 5470 to (34.67, -72.86, -8.25) mm, rotated rx 180 ry 0 rz 90 deg; joints [71.848, -16.33, 80.26, 0, 26.07, 71.848] to (46.33, -72.54, -8.25) mm, rotated rx 180 ry 0 rz 90 deg; joints [71.975, -16.086, 79.408, 0, 26.678, 71.975]
  MoveC 5471 to (47.86, -71.28, -8.25) mm, rotated rx 180 ry 0 rz 90 deg; joints [72.029, -16.062, 79.325, 0, 26.737, 72.029] to (48.8, -69.55, -8.25) mm, rotated rx 180 ry 0 rz 90 deg; joints [72.092, -16.054, 79.296, 0, 26.758, 72.092]
  MoveC 5472 to (49.27, -67.47, -8.25) mm, rotated rx -180 ry 0 rz 90 deg; joints [72.161, -16.058, 79.312, 0, 26.747, 72.161] to (48.8, -65.38, -8.25) mm, rotated rx 180 ry 0 rz 90 deg; joints [72.221, -16.083, 79.396, 0, 26.687, 72.221]
  MoveC 5473 to (36.99, -51.35, -8.25) mm, rotated rx 180 ry 0 rz 90 deg; joints [72.54, -16.425, 80.598, 0, 25.828, 72.54] to (25.12, -37.37, -8.25) mm, rotated rx 180 ry 0 rz 90 deg; joints [72.862, -16.755, 81.782, 0, 24.973, 72.862]
  MoveC 5474 to (24.85, -37.08, -8.25) mm, rotated rx 180 ry 0 rz 90 deg; joints [72.869, -16.762, 81.809, 0, 24.954, 72.869] to (24.55, -36.82, -8.25) mm, rotated rx -180 ry 0 rz 90 deg; joints [72.874, -16.77, 81.836, 0, 24.934, 72.874]
  MoveL 5475 to (22.97, -35.54, -8.25) mm, rotated rx 180 ry 0 rz 90 deg; joints [72.899, -16.809, 81.979, 0, 24.83, 72.899]
  MoveL 5476 to (12.79, -27.32, -8.25) mm, rotated rx 180 ry 0 rz 90 deg; joints [73.061, -17.057, 82.894, 0, 24.163, 73.061]
  MoveL 5477 to (12.37, -27.01, -8.25) mm, rotated rx 180 ry 0 rz 90 deg; joints [73.067, -17.067, 82.932, 0, 24.136, 73.067]
  MoveC 5478 to (10.48, -26.57, -8.25) mm, rotated rx 180 ry 0 rz 90 deg; joints [73.062, -17.106, 83.077, 0, 24.03, 73.062] to (8.59, -27.01, -8.25) mm, rotated rx -180 ry 0 rz 90 deg; joints [73.03, -17.14, 83.202, 0, 23.937, 73.03]
  MoveL 5479 to (8.18, -27.21, -8.25) mm, rotated rx -180 ry 0 rz 90 deg; joints [73.019, -17.146, 83.227, 0, 23.919, 73.019]
  MoveC 5480 to (7.29, -27.94, -8.25) mm, rotated rx 180 ry 0 rz 90 deg; joints [72.988, -17.159, 83.275, 0, 23.884, 72.988] to (6.76, -28.97, -8.25) mm, rotated rx -180 ry 0 rz 90 deg; joints [72.95, -17.163, 83.29, 0, 23.873, 72.95]
  MoveL 5481 to (-3.98, -69, -8.25) mm, rotated rx -180 ry 0 rz 90 deg; joints [71.569, -17.124, 83.143, 0, 23.981, 71.569]
  MoveC 5482 to (-4.02, -70.59, -8.25) mm, rotated rx -180 ry 0 rz 90 deg; joints [71.518, -17.115, 83.108, 0, 24.007, 71.518] to (-3.32, -72.02, -8.25) mm, rotated rx -180 ry 0 rz 90 deg; joints [71.48, -17.092, 83.024, 0, 24.068, 71.48]
  MoveC 5483 to (-2, -73.17, -8.25) mm, rotated rx 180 ry 0 rz 90 deg; joints [71.458, -17.06, 82.903, 0, 24.156, 71.458] to (-0.3, -73.57, -8.25) mm, rotated rx 180 ry 0 rz 90 deg; joints [71.463, -17.025, 82.773, 0, 24.252, 71.463]
  MoveC 5484 to (11.36, -73.38, -8.25) mm, rotated rx -180 ry 0 rz 90 deg; joints [71.592, -16.799, 81.943, 0, 24.856, 71.592] to (23.02, -73.14, -8.25) mm, rotated rx 180 ry 0 rz 90 deg; joints [71.72, -16.568, 81.105, 0, 25.462, 71.72]
  MoveL 5485 to (22.85, -65.59, -8.25) mm, rotated rx 180 ry 0 rz 90 deg; joints [71.954, -16.621, 81.297, 0, 25.324, 71.954]
  MoveL 5486 to (22.85, -65.59, -5.25) mm, rotated rx 180 ry 0 rz 90 deg; joints [71.954, -16.773, 81.399, 0, 25.373, 71.954]
  Establecer velocidad (1000.0 mm/s)
  MoveL 5487 to (22.85, -65.59, 10) mm, rotated rx -180 ry 0 rz 90 deg; joints [71.954, -17.543, 81.911, 0, 25.632, 71.954]
  Establecer velocidad (66.7 mm/s)
  MoveL 5488 to (-35.82, -51.71, 10) mm, rotated rx -180 ry 0 rz 90 deg; joints [71.784, -18.742, 86.384, 0, 22.359, 71.784]
  MoveL 5489 to (-35.82, -51.71, -5) mm, rotated rx 180 ry 0 rz 90 deg; joints [71.784, -17.971, 85.883, 0, 22.088, 71.784]
  MoveL 5490 to (-34.41, -52.27, -5.41) mm, rotated rx 180 ry 0 rz 90 deg; joints [71.781, -17.923, 85.759, 0, 22.164, 71.781]
  MoveL 5491 to (-32.9, -52.47, -5.81) mm, rotated rx -180 ry 0 rz 90 deg; joints [71.791, -17.874, 85.637, 0, 22.238, 71.791]
  MoveL 5492 to (-31.39, -52.34, -6.22) mm, rotated rx -180 ry 0 rz 90 deg; joints [71.811, -17.828, 85.521, 0, 22.307, 71.811]
  MoveL 5493 to (-29.94, -51.87, -6.62) mm, rotated rx -180 ry 0 rz 90 deg; joints [71.841, -17.784, 85.418, 0, 22.367, 71.841]
  MoveL 5494 to (-28.63, -51.1, -7.03) mm, rotated rx 180 ry 0 rz 90 deg; joints [71.88, -17.745, 85.331, 0, 22.414, 71.88]
  MoveL 5495 to (-27.53, -50.05, -7.44) mm, rotated rx -180 ry 0 rz 90 deg; joints [71.925, -17.711, 85.264, 0, 22.447, 71.925]
  MoveL 5496 to (-26.69, -48.79, -7.84) mm, rotated rx 180 ry 0 rz 90 deg; joints [71.975, -17.682, 85.22, 0, 22.462, 71.975]
  MoveL 5497 to (-26.17, -47.36, -8.25) mm, rotated rx 180 ry 0 rz 90 deg; joints [72.026, -17.66, 85.203, 0, 22.458, 72.026]
  MoveL 5498 to (-19.93, -23.4, -8.25) mm, rotated rx -180 ry 0 rz 90 deg; joints [72.865, -17.684, 85.296, 0, 22.388, 72.865]
  MoveC 5499 to (-19.86, -22.87, -8.25) mm, rotated rx 180 ry 0 rz 90 deg; joints [72.883, -17.686, 85.303, 0, 22.383, 72.883] to (-19.94, -22.34, -8.25) mm, rotated rx -180 ry 0 rz 90 deg; joints [72.899, -17.69, 85.32, 0, 22.37, 72.899]
  MoveC 5500 to (-20.86, -20.6, -8.25) mm, rotated rx -180 ry 0 rz 90 deg; joints [72.946, -17.716, 85.421, 0, 22.294, 72.946] to (-22.44, -19.43, -8.25) mm, rotated rx -180 ry 0 rz 90 deg; joints [72.969, -17.75, 85.556, 0, 22.193, 72.969]
  MoveC 5501 to (-23.2, -19.23, -8.25) mm, rotated rx -180 ry 0 rz 90 deg; joints [72.968, -17.764, 85.614, 0, 22.15, 72.968] to (-23.99, -19.27, -8.25) mm, rotated rx 180 ry 0 rz 90 deg; joints [72.958, -17.778, 85.668, 0, 22.11, 72.958]
  MoveL 5502 to (-32.69, -21.1, -8.25) mm, rotated rx 180 ry 0 rz 90 deg; joints [72.811, -17.918, 86.232, 0, 21.686, 72.811]
  MoveL 5503 to (-71.85, -29.4, -8.25) mm, rotated rx -180 ry 0 rz 90 deg; joints [72.131, -18.511, 88.719, 0, 19.792, 72.131]
  MoveC 5504 to (-73.74, -30.56, -8.25) mm, rotated rx 180 ry 0 rz 90 deg; joints [72.072, -18.534, 88.821, 0, 19.713, 72.072] to (-74.49, -32.66, -8.25) mm, rotated rx 180 ry 0 rz 90 deg; joints [71.994, -18.535, 88.825, 0, 19.71, 71.994]
  MoveL 5505 to (-74.49, -70.6, -8.25) mm, rotated rx -180 ry 0 rz 90 deg; joints [70.743, -18.336, 87.968, 0, 20.368, 70.743]
  MoveC 5506 to (-73.62, -72.77, -8.25) mm, rotated rx -180 ry 0 rz 90 deg; joints [70.682, -18.311, 87.859, 0, 20.452, 70.682] to (-71.55, -73.85, -8.25) mm, rotated rx -180 ry 0 rz 90 deg; joints [70.671, -18.272, 87.695, 0, 20.577, 70.671]
  MoveC 5507 to (-63.49, -73.83, -8.25) mm, rotated rx 180 ry 0 rz 90 deg; joints [70.763, -18.142, 87.152, 0, 20.99, 70.763] to (-55.44, -73.76, -8.25) mm, rotated rx 180 ry 0 rz 90 deg; joints [70.856, -18.01, 86.607, 0, 21.403, 70.856]
  MoveL 5508 to (-35.53, -73.57, -8.25) mm, rotated rx 180 ry 0 rz 90 deg; joints [71.083, -17.671, 85.246, 0, 22.425, 71.083]
  MoveC 5509 to (-33.62, -72.94, -8.25) mm, rotated rx 180 ry 0 rz 90 deg; joints [71.125, -17.641, 85.128, 0, 22.513, 71.125] to (-32.43, -71.32, -8.25) mm, rotated rx 180 ry 0 rz 90 deg; joints [71.19, -17.63, 85.084, 0, 22.546, 71.19]
  MoveC 5510 to (-32.35, -71.09, -8.25) mm, rotated rx 180 ry 0 rz 90 deg; joints [71.198, -17.63, 85.084, 0, 22.546, 71.198] to (-32.29, -70.86, -8.25) mm, rotated rx -180 ry 0 rz 90 deg; joints [71.206, -17.631, 85.085, 0, 22.545, 71.206]
  MoveL 5511 to (-26.17, -47.36, -8.25) mm, rotated rx 180 ry 0 rz 90 deg; joints [72.026, -17.66, 85.203, 0, 22.458, 72.026]
  MoveL 5512 to (-33.48, -45.46, -8.25) mm, rotated rx -180 ry 0 rz 90 deg; joints [72.011, -17.799, 85.752, 0, 22.046, 72.011]
  MoveL 5513 to (-33.48, -45.46, -5.25) mm, rotated rx 180 ry 0 rz 90 deg; joints [72.011, -17.953, 85.854, 0, 22.099, 72.011]
  Establecer velocidad (1000.0 mm/s)
  MoveL 5514 to (-33.48, -45.46, 10) mm, rotated rx 180 ry 0 rz 90 deg; joints [72.011, -18.737, 86.363, 0, 22.374, 72.011]
  Establecer velocidad (66.7 mm/s)
  MoveL 5515 to (-66.25, 35.99, 10) mm, rotated rx 180 ry 0 rz 90 deg; joints [74.382, -19.679, 90.275, 0, 19.404, 74.382]
  MoveL 5516 to (-66.25, 35.99, -5) mm, rotated rx 180 ry 0 rz 90 deg; joints [74.382, -18.894, 89.774, 0, 19.121, 74.382]
  MoveL 5517 to (-67.75, 36.17, -5.41) mm, rotated rx 180 ry 0 rz 90 deg; joints [74.374, -18.896, 89.864, 0, 19.032, 74.374]
  MoveL 5518 to (-69.26, 35.99, -5.81) mm, rotated rx 180 ry 0 rz 90 deg; joints [74.353, -18.897, 89.948, 0, 18.948, 74.353]
  MoveL 5519 to (-70.69, 35.48, -6.22) mm, rotated rx -180 ry 0 rz 90 deg; joints [74.322, -18.894, 90.021, 0, 18.873, 74.322]
  MoveL 5520 to (-71.97, 34.66, -6.62) mm, rotated rx -180 ry 0 rz 90 deg; joints [74.282, -18.888, 90.078, 0, 18.811, 74.282]
  MoveL 5521 to (-73.04, 33.58, -7.03) mm, rotated rx -180 ry 0 rz 90 deg; joints [74.235, -18.878, 90.115, 0, 18.763, 74.235]
  MoveL 5522 to (-73.85, 32.3, -7.44) mm, rotated rx 180 ry 0 rz 90 deg; joints [74.184, -18.864, 90.131, 0, 18.733, 74.184]
  MoveL 5523 to (-74.35, 30.86, -7.84) mm, rotated rx -180 ry 0 rz 90 deg; joints [74.13, -18.844, 90.123, 0, 18.72, 74.13]
  MoveL 5524 to (-74.49, 29.35, -8.25) mm, rotated rx 180 ry 0 rz 90 deg; joints [74.077, -18.818, 90.09, 0, 18.728, 74.077]
  MoveL 5525 to (-74.49, 1.42, -8.25) mm, rotated rx 180 ry 0 rz 90 deg; joints [73.133, -18.697, 89.541, 0, 19.156, 73.133]
  MoveL 5526 to (-74.44, 0.47, -8.25) mm, rotated rx 180 ry 0 rz 90 deg; joints [73.102, -18.692, 89.518, 0, 19.173, 73.102]
  MoveC 5527 to (-73.22, -1.45, -8.25) mm, rotated rx -180 ry 0 rz 90 deg; joints [73.05, -18.665, 89.397, 0, 19.267, 73.05] to (-71.07, -2.25, -8.25) mm, rotated rx 180 ry 0 rz 90 deg; joints [73.045, -18.629, 89.238, 0, 19.391, 73.045]
  MoveL 5528 to (-70.6, -2.19, -8.25) mm, rotated rx 180 ry 0 rz 90 deg; joints [73.052, -18.622, 89.207, 0, 19.415, 73.052]
  MoveC 5529 to (-67.28, -1.45, -8.25) mm, rotated rx 180 ry 0 rz 90 deg; joints [73.111, -18.575, 89, 0, 19.575, 73.111] to (-63.97, -0.68, -8.25) mm, rotated rx -180 ry 0 rz 90 deg; joints [73.17, -18.528, 88.792, 0, 19.735, 73.17]
  MoveC 5530 to (-42.88, 4.17, -8.25) mm, rotated rx 180 ry 0 rz 90 deg; joints [73.541, -18.216, 87.458, 0, 20.758, 73.541] to (-21.8, 9.05, -8.25) mm, rotated rx -180 ry 0 rz 90 deg; joints [73.904, -17.886, 86.101, 0, 21.784, 73.904]
  MoveC 5531 to (-19.38, 10.78, -8.25) mm, rotated rx 180 ry 0 rz 90 deg; joints [73.984, -17.853, 85.968, 0, 21.885, 73.984] to (-19.13, 13.74, -8.25) mm, rotated rx -180 ry 0 rz 90 deg; joints [74.083, -17.863, 86.009, 0, 21.854, 74.083]
  MoveL 5532 to (-25.67, 32.05, -8.25) mm, rotated rx 180 ry 0 rz 90 deg; joints [74.627, -18.062, 86.821, 0, 21.241, 74.627]
  MoveC 5533 to (-26.09, 32.85, -8.25) mm, rotated rx -180 ry 0 rz 90 deg; joints [74.649, -18.073, 86.865, 0, 21.208, 74.649] to (-26.71, 33.51, -8.25) mm, rotated rx 180 ry 0 rz 90 deg; joints [74.665, -18.087, 86.921, 0, 21.166, 74.665]
  MoveL 5534 to (-27.01, 33.74, -8.25) mm, rotated rx 180 ry 0 rz 90 deg; joints [74.67, -18.093, 86.945, 0, 21.147, 74.67]
  MoveC 5535 to (-48.16, 47.34, -8.25) mm, rotated rx 180 ry 0 rz 90 deg; joints [74.933, -18.495, 88.651, 0, 19.844, 74.933] to (-69.33, 60.9, -8.25) mm, rotated rx -180 ry 0 rz 90 deg; joints [75.201, -18.869, 90.325, 0, 18.545, 75.201]
  MoveC 5536 to (-70.55, 61.31, -8.25) mm, rotated rx 180 ry 0 rz 90 deg; joints [75.204, -18.888, 90.413, 0, 18.475, 75.204] to (-71.82, 61.12, -8.25) mm, rotated rx 180 ry 0 rz 90 deg; joints [75.186, -18.906, 90.495, 0, 18.411, 75.186]
  MoveC 5537 to (-73.38, 60.28, -8.25) mm, rotated rx 180 ry 0 rz 90 deg; joints [75.143, -18.925, 90.584, 0, 18.341, 75.143] to (-74.39, 58.83, -8.25) mm, rotated rx 180 ry 0 rz 90 deg; joints [75.084, -18.934, 90.626, 0, 18.308, 75.084]
  MoveC 5538 to (-74.46, 58.53, -8.25) mm, rotated rx 180 ry 0 rz 90 deg; joints [75.073, -18.934, 90.626, 0, 18.308, 75.073] to (-74.49, 58.23, -8.25) mm, rotated rx -180 ry 0 rz 90 deg; joints [75.063, -18.933, 90.622, 0, 18.312, 75.063]
  MoveL 5539 to (-74.49, 29.35, -8.25) mm, rotated rx 180 ry 0 rz 90 deg; joints [74.077, -18.818, 90.09, 0, 18.728, 74.077]
  MoveL 5540 to (-66.94, 29.35, -8.25) mm, rotated rx 180 ry 0 rz 90 deg; joints [74.15, -18.706, 89.584, 0, 19.122, 74.15]
  MoveL 5541 to (-66.94, 29.35, -5.25) mm, rotated rx 180 ry 0 rz 90 deg; joints [74.15, -18.863, 89.686, 0, 19.177, 74.15]
  Establecer velocidad (1000.0 mm/s)
  MoveL 5542 to (-66.94, 29.35, 10) mm, rotated rx 180 ry 0 rz 90 deg; joints [74.15, -19.661, 90.195, 0, 19.466, 74.15]
  Establecer velocidad (66.7 mm/s)
  MoveL 5543 to (-66.08, 35.99, 10) mm, rotated rx 180 ry 0 rz 90 deg; joints [74.383, -19.676, 90.263, 0, 19.413, 74.383]
  MoveL 5544 to (-66.08, 35.99, -5.25) mm, rotated rx 180 ry 0 rz 90 deg; joints [74.383, -18.879, 89.754, 0, 19.125, 74.383]
  MoveL 5545 to (-67.58, 36.17, -5.66) mm, rotated rx 180 ry 0 rz 90 deg; joints [74.375, -18.881, 89.845, 0, 19.036, 74.375]
  MoveL 5546 to (-69.09, 35.99, -6.06) mm, rotated rx 180 ry 0 rz 90 deg; joints [74.355, -18.881, 89.929, 0, 18.952, 74.355]
  MoveL 5547 to (-70.52, 35.48, -6.47) mm, rotated rx 180 ry 0 rz 90 deg; joints [74.324, -18.879, 90.001, 0, 18.877, 74.324]
  MoveL 5548 to (-71.81, 34.66, -6.88) mm, rotated rx 180 ry 0 rz 90 deg; joints [74.284, -18.873, 90.058, 0, 18.815, 74.284]
  MoveL 5549 to (-72.88, 33.58, -7.28) mm, rotated rx 180 ry 0 rz 90 deg; joints [74.237, -18.863, 90.095, 0, 18.768, 74.237]
  MoveL 5550 to (-73.68, 32.3, -7.69) mm, rotated rx 180 ry 0 rz 90 deg; joints [74.185, -18.848, 90.111, 0, 18.737, 74.185]
  MoveL 5551 to (-74.18, 30.86, -8.09) mm, rotated rx 180 ry 0 rz 90 deg; joints [74.132, -18.828, 90.103, 0, 18.725, 74.132]
  MoveL 5552 to (-74.32, 29.35, -8.5) mm, rotated rx 180 ry 0 rz 90 deg; joints [74.079, -18.802, 90.07, 0, 18.732, 74.079]
  MoveL 5553 to (-74.32, 2.37, -8.5) mm, rotated rx 180 ry 0 rz 90 deg; joints [73.167, -18.685, 89.54, 0, 19.145, 73.167]
  MoveL 5554 to (-74.32, 1.42, -8.5) mm, rotated rx -180 ry 0 rz 90 deg; joints [73.135, -18.681, 89.521, 0, 19.16, 73.135]
  MoveC 5555 to (-73.23, -1.15, -8.5) mm, rotated rx -180 ry 0 rz 90 deg; joints [73.06, -18.653, 89.396, 0, 19.257, 73.06] to (-70.58, -2.03, -8.5) mm, rotated rx -180 ry 0 rz 90 deg; joints [73.057, -18.609, 89.2, 0, 19.409, 73.057]
  MoveC 5556 to (-70.42, -2.01, -8.5) mm, rotated rx 180 ry 0 rz 90 deg; joints [73.06, -18.607, 89.19, 0, 19.416, 73.06] to (-70.27, -1.98, -8.5) mm, rotated rx 180 ry 0 rz 90 deg; joints [73.062, -18.605, 89.181, 0, 19.424, 73.062]
  MoveL 5557 to (-27.01, 8, -8.5) mm, rotated rx -180 ry 0 rz 90 deg; joints [73.821, -17.957, 86.434, 0, 21.523, 73.821]
  MoveL 5558 to (-21.8, 9.22, -8.5) mm, rotated rx -180 ry 0 rz 90 deg; joints [73.91, -17.874, 86.096, 0, 21.777, 73.91]
  MoveC 5559 to (-19.55, 10.93, -8.5) mm, rotated rx -180 ry 0 rz 90 deg; joints [73.987, -17.844, 85.974, 0, 21.869, 73.987] to (-19.3, 13.74, -8.5) mm, rotated rx 180 ry 0 rz 90 deg; joints [74.082, -17.853, 86.013, 0, 21.84, 74.082]
  MoveL 5560 to (-19.43, 14.08, -8.5) mm, rotated rx -180 ry 0 rz 90 deg; joints [74.092, -17.857, 86.028, 0, 21.829, 74.092]
  MoveL 5561 to (-25.73, 31.75, -8.5) mm, rotated rx -180 ry 0 rz 90 deg; joints [74.616, -18.049, 86.811, 0, 21.238, 74.616]
  MoveL 5562 to (-26.06, 32.46, -8.5) mm, rotated rx 180 ry 0 rz 90 deg; joints [74.636, -18.058, 86.847, 0, 21.211, 74.636]
  MoveC 5563 to (-26.52, 33.13, -8.5) mm, rotated rx -180 ry 0 rz 90 deg; joints [74.654, -18.069, 86.892, 0, 21.177, 74.654] to (-27.15, 33.64, -8.5) mm, rotated rx -180 ry 0 rz 90 deg; joints [74.666, -18.082, 86.945, 0, 21.137, 74.666]
  MoveC 5564 to (-48.23, 47.2, -8.5) mm, rotated rx -180 ry 0 rz 90 deg; joints [74.927, -18.483, 88.645, 0, 19.838, 74.927] to (-69.33, 60.71, -8.5) mm, rotated rx 180 ry 0 rz 90 deg; joints [75.195, -18.855, 90.313, 0, 18.542, 75.195]
  MoveC 5565 to (-69.91, 60.97, -8.5) mm, rotated rx 180 ry 0 rz 90 deg; joints [75.199, -18.865, 90.356, 0, 18.509, 75.199] to (-70.54, 61.06, -8.5) mm, rotated rx 180 ry 0 rz 90 deg; joints [75.196, -18.874, 90.4, 0, 18.474, 75.196]
  MoveC 5566 to (-72.45, 60.57, -8.5) mm, rotated rx 180 ry 0 rz 90 deg; joints [75.162, -18.9, 90.519, 0, 18.381, 75.162] to (-73.91, 59.25, -8.5) mm, rotated rx 180 ry 0 rz 90 deg; joints [75.103, -18.916, 90.593, 0, 18.323, 75.103]
  MoveC 5567 to (-74.21, 58.61, -8.5) mm, rotated rx 180 ry 0 rz 90 deg; joints [75.079, -18.918, 90.602, 0, 18.316, 75.079] to (-74.32, 57.92, -8.5) mm, rotated rx 180 ry 0 rz 90 deg; joints [75.054, -18.917, 90.597, 0, 18.32, 75.054]
  MoveL 5568 to (-74.32, 29.35, -8.5) mm, rotated rx 180 ry 0 rz 90 deg; joints [74.079, -18.802, 90.07, 0, 18.732, 74.079]
  MoveL 5569 to (-66.77, 29.35, -8.5) mm, rotated rx 180 ry 0 rz 90 deg; joints [74.152, -18.691, 89.564, 0, 19.126, 74.152]
  MoveL 5570 to (-66.77, 29.35, -5.5) mm, rotated rx -180 ry 0 rz 90 deg; joints [74.152, -18.848, 89.666, 0, 19.182, 74.152]
  Establecer velocidad (1000.0 mm/s)
  MoveL 5571 to (-66.77, 29.35, 10) mm, rotated rx -180 ry 0 rz 90 deg; joints [74.152, -19.658, 90.184, 0, 19.475, 74.152]
  Establecer velocidad (66.7 mm/s)
  MoveL 5572 to (-39.5, -31.11, 10) mm, rotated rx 180 ry 0 rz 90 deg; joints [72.415, -18.922, 87.096, 0, 21.826, 72.415]
  MoveL 5573 to (-39.5, -31.11, -5.25) mm, rotated rx -180 ry 0 rz 90 deg; joints [72.415, -18.135, 86.587, 0, 21.549, 72.415]
  MoveL 5574 to (-39.63, -29.6, -5.66) mm, rotated rx -180 ry 0 rz 90 deg; joints [72.463, -18.125, 86.615, 0, 21.51, 72.463]
  MoveL 5575 to (-40.13, -28.16, -6.06) mm, rotated rx -180 ry 0 rz 90 deg; joints [72.505, -18.12, 86.667, 0, 21.453, 72.505]
  MoveL 5576 to (-40.93, -26.87, -6.47) mm, rotated rx -180 ry 0 rz 90 deg; joints [72.539, -18.119, 86.736, 0, 21.383, 72.539]
  MoveL 5577 to (-41.99, -25.79, -6.88) mm, rotated rx -180 ry 0 rz 90 deg; joints [72.563, -18.122, 86.819, 0, 21.303, 72.563]
  MoveL 5578 to (-43.27, -24.97, -7.28) mm, rotated rx 180 ry 0 rz 90 deg; joints [72.577, -18.126, 86.91, 0, 21.216, 72.577]
  MoveL 5579 to (-44.7, -24.46, -7.69) mm, rotated rx -180 ry 0 rz 90 deg; joints [72.579, -18.132, 87.005, 0, 21.126, 72.579]
  MoveL 5580 to (-46.21, -24.27, -8.09) mm, rotated rx 180 ry 0 rz 90 deg; joints [72.57, -18.136, 87.099, 0, 21.038, 72.57]
  MoveL 5581 to (-47.72, -24.45, -8.5) mm, rotated rx 180 ry 0 rz 90 deg; joints [72.548, -18.139, 87.184, 0, 20.955, 72.548]
  MoveL 5582 to (-47.86, -24.48, -8.5) mm, rotated rx 180 ry 0 rz 90 deg; joints [72.546, -18.141, 87.193, 0, 20.948, 72.546]
  MoveL 5583 to (-71.73, -29.54, -8.5) mm, rotated rx 180 ry 0 rz 90 deg; joints [72.128, -18.495, 88.7, 0, 19.796, 72.128]
  MoveC 5584 to (-73.5, -30.58, -8.5) mm, rotated rx -180 ry 0 rz 90 deg; joints [72.074, -18.517, 88.796, 0, 19.721, 72.074] to (-74.3, -32.47, -8.5) mm, rotated rx -180 ry 0 rz 90 deg; joints [72.002, -18.52, 88.808, 0, 19.712, 72.002]
  MoveL 5585 to (-74.31, -32.69, -8.5) mm, rotated rx 180 ry 0 rz 90 deg; joints [71.995, -18.519, 88.804, 0, 19.715, 71.995]
  MoveL 5586 to (-74.32, -33.64, -8.5) mm, rotated rx 180 ry 0 rz 90 deg; joints [71.963, -18.515, 88.784, 0, 19.731, 71.963]
  MoveL 5587 to (-74.32, -69.65, -8.5) mm, rotated rx 180 ry 0 rz 90 deg; joints [70.776, -18.326, 87.971, 0, 20.356, 70.776]
  MoveL 5588 to (-74.31, -70.6, -8.5) mm, rotated rx -180 ry 0 rz 90 deg; joints [70.745, -18.321, 87.948, 0, 20.373, 70.745]
  MoveC 5589 to (-73.47, -72.62, -8.5) mm, rotated rx -180 ry 0 rz 90 deg; joints [70.689, -18.296, 87.844, 0, 20.452, 70.689] to (-71.55, -73.68, -8.5) mm, rotated rx -180 ry 0 rz 90 deg; joints [70.676, -18.26, 87.69, 0, 20.57, 70.676]
  MoveL 5590 to (-70.6, -73.71, -8.5) mm, rotated rx -180 ry 0 rz 90 deg; joints [70.686, -18.245, 87.625, 0, 20.619, 70.686]
  MoveL 5591 to (-36.48, -73.41, -8.5) mm, rotated rx -180 ry 0 rz 90 deg; joints [71.078, -17.676, 85.307, 0, 22.369, 71.078]
  MoveL 5592 to (-35.59, -73.4, -8.5) mm, rotated rx 180 ry 0 rz 90 deg; joints [71.088, -17.66, 85.245, 0, 22.415, 71.088]
  MoveC 5593 to (-33.74, -72.79, -8.5) mm, rotated rx 180 ry 0 rz 90 deg; joints [71.128, -17.632, 85.132, 0, 22.5, 71.128] to (-32.57, -71.24, -8.5) mm, rotated rx 180 ry 0 rz 90 deg; joints [71.191, -17.62, 85.087, 0, 22.533, 71.191]
  MoveC 5594 to (-32.5, -71.02, -8.5) mm, rotated rx 180 ry 0 rz 90 deg; joints [71.199, -17.62, 85.088, 0, 22.533, 71.199] to (-32.43, -70.79, -8.5) mm, rotated rx 180 ry 0 rz 90 deg; joints [71.207, -17.621, 85.088, 0, 22.532, 71.207]
  MoveL 5595 to (-20.37, -24.48, -8.5) mm, rotated rx -180 ry 0 rz 90 deg; joints [72.825, -17.673, 85.295, 0, 22.378, 72.825]
  MoveL 5596 to (-20.07, -23.22, -8.5) mm, rotated rx 180 ry 0 rz 90 deg; joints [72.869, -17.675, 85.301, 0, 22.374, 72.869]
  MoveC 5597 to (-21.19, -20.65, -8.5) mm, rotated rx -180 ry 0 rz 90 deg; joints [72.941, -17.708, 85.434, 0, 22.274, 72.941] to (-23.69, -19.41, -8.5) mm, rotated rx -180 ry 0 rz 90 deg; joints [72.957, -17.759, 85.635, 0, 22.123, 72.957]
  MoveL 5598 to (-24.17, -19.48, -8.5) mm, rotated rx -180 ry 0 rz 90 deg; joints [72.95, -17.767, 85.667, 0, 22.1, 72.95]
  MoveL 5599 to (-45.01, -23.87, -8.5) mm, rotated rx 180 ry 0 rz 90 deg; joints [72.595, -18.098, 87.012, 0, 21.086, 72.595]
  MoveL 5600 to (-47.72, -24.45, -8.5) mm, rotated rx 180 ry 0 rz 90 deg; joints [72.548, -18.139, 87.184, 0, 20.955, 72.548]
  MoveL 5601 to (-46.13, -31.83, -8.5) mm, rotated rx -180 ry 0 rz 90 deg; joints [72.323, -18.075, 86.916, 0, 21.159, 72.323]
  MoveL 5602 to (-46.13, -31.83, -5.5) mm, rotated rx -180 ry 0 rz 90 deg; joints [72.323, -18.23, 87.018, 0, 21.212, 72.323]
  Establecer velocidad (1000.0 mm/s)
  MoveL 5603 to (-46.13, -31.83, 10) mm, rotated rx 180 ry 0 rz 90 deg; joints [72.323, -19.031, 87.535, 0, 21.495, 72.323]
  Establecer velocidad (66.7 mm/s)
  MoveL 5604 to (15.86, -64.84, 10) mm, rotated rx -180 ry 0 rz 90 deg; joints [71.906, -17.69, 82.435, 0, 25.255, 71.906]
  MoveL 5605 to (15.86, -64.84, -5.25) mm, rotated rx 180 ry 0 rz 90 deg; joints [71.906, -16.918, 81.924, 0, 24.994, 71.906]
  MoveL 5606 to (15.71, -66.35, -5.66) mm, rotated rx 180 ry 0 rz 90 deg; joints [71.857, -16.891, 81.885, 0, 25.006, 71.857]
  MoveL 5607 to (15.93, -67.85, -6.06) mm, rotated rx 180 ry 0 rz 90 deg; joints [71.812, -16.856, 81.82, 0, 25.036, 71.812]
  MoveL 5608 to (16.47, -69.27, -6.47) mm, rotated rx -180 ry 0 rz 90 deg; joints [71.773, -16.815, 81.733, 0, 25.082, 71.773]
  MoveL 5609 to (17.32, -70.54, -6.88) mm, rotated rx 180 ry 0 rz 90 deg; joints [71.742, -16.769, 81.628, 0, 25.141, 71.742]
  MoveL 5610 to (18.42, -71.58, -7.28) mm, rotated rx 180 ry 0 rz 90 deg; joints [71.721, -16.72, 81.509, 0, 25.21, 71.721]
  MoveL 5611 to (19.73, -72.36, -7.69) mm, rotated rx -180 ry 0 rz 90 deg; joints [71.71, -16.668, 81.382, 0, 25.286, 71.71]
  MoveL 5612 to (21.17, -72.82, -8.09) mm, rotated rx -180 ry 0 rz 90 deg; joints [71.711, -16.615, 81.252, 0, 25.363, 71.711]
  MoveL 5613 to (22.68, -72.93, -8.5) mm, rotated rx -180 ry 0 rz 90 deg; joints [71.723, -16.563, 81.126, 0, 25.437, 71.723]
  MoveC 5614 to (34.26, -72.63, -8.5) mm, rotated rx -180 ry 0 rz 90 deg; joints [71.851, -16.328, 80.288, 0, 26.04, 71.851] to (45.84, -72.29, -8.5) mm, rotated rx 180 ry 0 rz 90 deg; joints [71.978, -16.086, 79.442, 0, 26.644, 71.978]
  MoveC 5615 to (48.32, -69.29, -8.5) mm, rotated rx -180 ry 0 rz 90 deg; joints [72.096, -16.053, 79.33, 0, 26.724, 72.096] to (48.46, -65.39, -8.5) mm, rotated rx 180 ry 0 rz 90 deg; joints [72.217, -16.078, 79.413, 0, 26.665, 72.217]
  MoveL 5616 to (44.07, -60.12, -8.5) mm, rotated rx -180 ry 0 rz 90 deg; joints [72.337, -16.207, 79.863, 0, 26.344, 72.337]
  MoveL 5617 to (25.11, -37.7, -8.5) mm, rotated rx 180 ry 0 rz 90 deg; joints [72.852, -16.741, 81.767, 0, 24.974, 72.852]
  MoveL 5618 to (24.87, -37.43, -8.5) mm, rotated rx 180 ry 0 rz 90 deg; joints [72.858, -16.747, 81.791, 0, 24.956, 72.858]
  MoveL 5619 to (23.79, -36.48, -8.5) mm, rotated rx -180 ry 0 rz 90 deg; joints [72.877, -16.774, 81.89, 0, 24.884, 72.877]
  MoveL 5620 to (12.69, -27.51, -8.5) mm, rotated rx -180 ry 0 rz 90 deg; joints [73.054, -17.046, 82.889, 0, 24.156, 73.054]
  MoveC 5621 to (10.03, -26.96, -8.5) mm, rotated rx -180 ry 0 rz 90 deg; joints [73.046, -17.1, 83.092, 0, 24.008, 73.046] to (7.58, -28.12, -8.5) mm, rotated rx 180 ry 0 rz 90 deg; joints [72.985, -17.14, 83.242, 0, 23.898, 72.985]
  MoveL 5622 to (7.11, -28.74, -8.5) mm, rotated rx 180 ry 0 rz 90 deg; joints [72.96, -17.145, 83.262, 0, 23.883, 72.96]
  MoveL 5623 to (7.04, -28.9, -8.5) mm, rotated rx 180 ry 0 rz 90 deg; joints [72.954, -17.146, 83.264, 0, 23.882, 72.954]
  MoveL 5624 to (-3.67, -68.7, -8.5) mm, rotated rx 180 ry 0 rz 90 deg; joints [71.581, -17.107, 83.12, 0, 23.988, 71.581]
  MoveL 5625 to (-3.77, -69.18, -8.5) mm, rotated rx 180 ry 0 rz 90 deg; joints [71.565, -17.106, 83.116, 0, 23.99, 71.565]
  MoveC 5626 to (-2.99, -71.95, -8.5) mm, rotated rx 180 ry 0 rz 90 deg; joints [71.486, -17.074, 82.994, 0, 24.079, 71.486] to (-0.47, -73.35, -8.5) mm, rotated rx 180 ry 0 rz 90 deg; joints [71.468, -17.017, 82.782, 0, 24.235, 71.468]
  MoveC 5627 to (11.11, -73.16, -8.5) mm, rotated rx -180 ry 0 rz 90 deg; joints [71.596, -16.793, 81.958, 0, 24.835, 71.596] to (22.68, -72.93, -8.5) mm, rotated rx -180 ry 0 rz 90 deg; joints [71.723, -16.563, 81.126, 0, 25.437, 71.723]
  MoveL 5628 to (22.51, -65.38, -8.5) mm, rotated rx 180 ry 0 rz 90 deg; joints [71.957, -16.617, 81.319, 0, 25.298, 71.957]
  MoveL 5629 to (22.51, -65.38, -5.5) mm, rotated rx 180 ry 0 rz 90 deg; joints [71.957, -16.769, 81.421, 0, 25.348, 71.957]
  Establecer velocidad (1000.0 mm/s)
  MoveL 5630 to (22.51, -65.38, 10) mm, rotated rx 180 ry 0 rz 90 deg; joints [71.957, -17.552, 81.941, 0, 25.611, 71.957]
  Establecer velocidad (66.7 mm/s)
  MoveL 5631 to (62.6, -31.7, 10) mm, rotated rx 180 ry 0 rz 90 deg; joints [73.395, -16.925, 79.76, 0, 27.165, 73.395]
  MoveL 5632 to (62.6, -31.7, -5.25) mm, rotated rx -180 ry 0 rz 90 deg; joints [73.395, -16.16, 79.246, 0, 26.914, 73.395]
  MoveL 5633 to (64.11, -31.89, -5.66) mm, rotated rx -180 ry 0 rz 90 deg; joints [73.403, -16.106, 79.115, 0, 26.991, 73.403]
  MoveL 5634 to (65.62, -31.7, -6.06) mm, rotated rx 180 ry 0 rz 90 deg; joints [73.422, -16.054, 78.992, 0, 27.062, 73.422]
  MoveL 5635 to (67.05, -31.19, -6.47) mm, rotated rx -180 ry 0 rz 90 deg; joints [73.452, -16.005, 78.882, 0, 27.123, 73.452]
  MoveL 5636 to (68.33, -30.38, -6.88) mm, rotated rx 180 ry 0 rz 90 deg; joints [73.489, -15.962, 78.79, 0, 27.172, 73.489]
  MoveL 5637 to (69.4, -29.3, -7.28) mm, rotated rx 180 ry 0 rz 90 deg; joints [73.532, -15.925, 78.719, 0, 27.206, 73.532]
  MoveL 5638 to (70.2, -28.01, -7.69) mm, rotated rx -180 ry 0 rz 90 deg; joints [73.579, -15.895, 78.673, 0, 27.222, 73.579]
  MoveL 5639 to (70.7, -26.57, -8.09) mm, rotated rx 180 ry 0 rz 90 deg; joints [73.628, -15.873, 78.654, 0, 27.22, 73.628]
  MoveL 5640 to (70.84, -25.06, -8.5) mm, rotated rx -180 ry 0 rz 90 deg; joints [73.676, -15.86, 78.663, 0, 27.197, 73.676]
  MoveL 5641 to (70.84, -17.43, -8.5) mm, rotated rx -180 ry 0 rz 90 deg; joints [73.912, -15.909, 78.83, 0, 27.079, 73.912]
  MoveC 5642 to (68.28, -14.15, -8.5) mm, rotated rx 180 ry 0 rz 90 deg; joints [73.991, -15.985, 79.094, 0, 26.891, 73.991] to (64.24, -13.13, -8.5) mm, rotated rx -180 ry 0 rz 90 deg; joints [73.987, -16.079, 79.419, 0, 26.66, 73.987]
  MoveL 5643 to (56.31, -23.88, -8.5) mm, rotated rx -180 ry 0 rz 90 deg; joints [73.58, -16.183, 79.779, 0, 26.404, 73.58]
  MoveC 5644 to (55.67, -26.01, -8.5) mm, rotated rx 180 ry 0 rz 90 deg; joints [73.508, -16.183, 79.78, 0, 26.403, 73.508] to (56.52, -28.06, -8.5) mm, rotated rx 180 ry 0 rz 90 deg; joints [73.451, -16.152, 79.671, 0, 26.481, 73.451]
  MoveL 5645 to (64.67, -37.11, -8.5) mm, rotated rx 180 ry 0 rz 90 deg; joints [73.246, -15.917, 78.858, 0, 27.059, 73.246]
  MoveC 5646 to (68.56, -36.02, -8.5) mm, rotated rx 180 ry 0 rz 90 deg; joints [73.316, -15.838, 78.59, 0, 27.249, 73.316] to (70.84, -32.69, -8.5) mm, rotated rx -180 ry 0 rz 90 deg; joints [73.44, -15.81, 78.492, 0, 27.318, 73.44]
  MoveL 5647 to (70.84, -25.06, -8.5) mm, rotated rx -180 ry 0 rz 90 deg; joints [73.676, -15.86, 78.663, 0, 27.197, 73.676]
  MoveL 5648 to (63.29, -25.06, -8.5) mm, rotated rx -180 ry 0 rz 90 deg; joints [73.607, -16.025, 79.231, 0, 26.794, 73.607]
  MoveL 5649 to (63.29, -25.06, -5.5) mm, rotated rx 180 ry 0 rz 90 deg; joints [73.607, -16.176, 79.334, 0, 26.842, 73.607]
  Establecer velocidad (1000.0 mm/s)
  MoveL 5650 to (63.29, -25.06, 10) mm, rotated rx 180 ry 0 rz 90 deg; joints [73.607, -16.953, 79.856, 0, 27.097, 73.607]
  Establecer velocidad (66.7 mm/s)
  MoveL 5651 to (35.82, 20.15, 10) mm, rotated rx 180 ry 0 rz 90 deg; joints [74.786, -17.8, 82.831, 0, 24.969, 74.786]
  MoveL 5652 to (35.82, 20.15, -5.25) mm, rotated rx 180 ry 0 rz 90 deg; joints [74.786, -17.027, 82.32, 0, 24.707, 74.786]
  MoveL 5653 to (35.98, 21.65, -5.66) mm, rotated rx 180 ry 0 rz 90 deg; joints [74.836, -17.011, 82.324, 0, 24.687, 74.836]
  MoveL 5654 to (35.78, 23.16, -6.06) mm, rotated rx -180 ry 0 rz 90 deg; joints [74.882, -17.003, 82.355, 0, 24.647, 74.882]
  MoveL 5655 to (35.25, 24.58, -6.47) mm, rotated rx -180 ry 0 rz 90 deg; joints [74.923, -17, 82.408, 0, 24.592, 74.923]
  MoveL 5656 to (34.41, 25.85, -6.88) mm, rotated rx 180 ry 0 rz 90 deg; joints [74.956, -17.003, 82.48, 0, 24.523, 74.956]
  MoveL 5657 to (33.31, 26.91, -7.28) mm, rotated rx 180 ry 0 rz 90 deg; joints [74.981, -17.009, 82.567, 0, 24.443, 74.981]
  MoveL 5658 to (32.01, 27.69, -7.69) mm, rotated rx -180 ry 0 rz 90 deg; joints [74.995, -17.018, 82.663, 0, 24.356, 74.995]
  MoveL 5659 to (30.57, 28.17, -8.09) mm, rotated rx -180 ry 0 rz 90 deg; joints [74.998, -17.028, 82.763, 0, 24.266, 74.998]
  MoveL 5660 to (29.06, 28.29, -8.5) mm, rotated rx -180 ry 0 rz 90 deg; joints [74.988, -17.038, 82.861, 0, 24.177, 74.988]
  MoveL 5661 to (11.85, 28.04, -8.5) mm, rotated rx 180 ry 0 rz 90 deg; joints [74.831, -17.365, 84.095, 0, 23.27, 74.831]
  MoveL 5662 to (10.9, 27.99, -8.5) mm, rotated rx 180 ry 0 rz 90 deg; joints [74.821, -17.382, 84.162, 0, 23.22, 74.821]
  MoveC 5663 to (8.49, 26.45, -8.5) mm, rotated rx -180 ry 0 rz 90 deg; joints [74.75, -17.419, 84.304, 0, 23.115, 74.75] to (7.75, 23.69, -8.5) mm, rotated rx 180 ry 0 rz 90 deg; joints [74.653, -17.419, 84.303, 0, 23.116, 74.653]
  MoveL 5664 to (7.89, 23.22, -8.5) mm, rotated rx 180 ry 0 rz 90 deg; joints [74.639, -17.414, 84.283, 0, 23.13, 74.639]
  MoveL 5665 to (12.74, 9.95, -8.5) mm, rotated rx 180 ry 0 rz 90 deg; joints [74.254, -17.254, 83.673, 0, 23.581, 74.254]
  MoveL 5666 to (12.79, 9.84, -8.5) mm, rotated rx 180 ry 0 rz 90 deg; joints [74.251, -17.252, 83.667, 0, 23.585, 74.251]
  MoveC 5667 to (13.19, 9.17, -8.5) mm, rotated rx -180 ry 0 rz 90 deg; joints [74.233, -17.241, 83.625, 0, 23.616, 74.233] to (13.74, 8.61, -8.5) mm, rotated rx 180 ry 0 rz 90 deg; joints [74.22, -17.228, 83.575, 0, 23.653, 74.22]
  MoveL 5668 to (14.44, 8.05, -8.5) mm, rotated rx 180 ry 0 rz 90 deg; joints [74.208, -17.212, 83.513, 0, 23.699, 74.208]
  MoveL 5669 to (28.42, -2.58, -8.5) mm, rotated rx 180 ry 0 rz 90 deg; joints [73.996, -16.883, 82.286, 0, 24.596, 73.996]
  MoveC 5670 to (29.05, -2.94, -8.5) mm, rotated rx 180 ry 0 rz 90 deg; joints [73.99, -16.868, 82.233, 0, 24.635, 73.99] to (29.75, -3.13, -8.5) mm, rotated rx 180 ry 0 rz 90 deg; joints [73.99, -16.853, 82.178, 0, 24.675, 73.99]
  MoveC 5671 to (32.04, -2.82, -8.5) mm, rotated rx 180 ry 0 rz 90 deg; joints [74.021, -16.809, 82.018, 0, 24.792, 74.021] to (33.83, -1.36, -8.5) mm, rotated rx -180 ry 0 rz 90 deg; joints [74.084, -16.782, 81.918, 0, 24.864, 74.084]
  MoveL 5672 to (49.11, 20.37, -8.5) mm, rotated rx -180 ry 0 rz 90 deg; joints [74.908, -16.595, 81.239, 0, 25.356, 74.908]
  MoveL 5673 to (50.1, 21.8, -8.5) mm, rotated rx -180 ry 0 rz 90 deg; joints [74.961, -16.582, 81.194, 0, 25.388, 74.961]
  MoveC 5674 to (49.85, 25.66, -8.5) mm, rotated rx 180 ry 0 rz 90 deg; joints [75.082, -16.609, 81.289, 0, 25.32, 75.082] to (47.22, 28.5, -8.5) mm, rotated rx -180 ry 0 rz 90 deg; joints [75.15, -16.678, 81.538, 0, 25.139, 75.15]
  MoveL 5675 to (40.27, 28.45, -8.5) mm, rotated rx -180 ry 0 rz 90 deg; joints [75.09, -16.818, 82.047, 0, 24.77, 75.09]
  MoveL 5676 to (29.06, 28.29, -8.5) mm, rotated rx -180 ry 0 rz 90 deg; joints [74.988, -17.038, 82.861, 0, 24.177, 74.988]
  MoveL 5677 to (29.17, 20.74, -8.5) mm, rotated rx -180 ry 0 rz 90 deg; joints [74.747, -16.996, 82.705, 0, 24.291, 74.747]
  MoveL 5678 to (29.17, 20.74, -5.5) mm, rotated rx 180 ry 0 rz 90 deg; joints [74.747, -17.149, 82.807, 0, 24.342, 74.747]
  Establecer velocidad (1000.0 mm/s)
  MoveL 5679 to (29.17, 20.74, 10) mm, rotated rx -180 ry 0 rz 90 deg; joints [74.747, -17.936, 83.326, 0, 24.61, 74.747]
  Establecer velocidad (66.7 mm/s)
  MoveL 5680 to (28.9, 64.3, 10) mm, rotated rx 180 ry 0 rz 90 deg; joints [76.15, -18.162, 84.164, 0, 23.999, 76.15]
  MoveL 5681 to (28.9, 64.3, -5.25) mm, rotated rx 180 ry 0 rz 90 deg; joints [76.15, -17.386, 83.654, 0, 23.732, 76.15]
  MoveL 5682 to (29.12, 65.8, -5.66) mm, rotated rx 180 ry 0 rz 90 deg; joints [76.201, -17.368, 83.651, 0, 23.717, 76.201]
  MoveL 5683 to (28.97, 67.31, -6.06) mm, rotated rx -180 ry 0 rz 90 deg; joints [76.249, -17.357, 83.674, 0, 23.682, 76.249]
  MoveL 5684 to (28.49, 68.75, -6.47) mm, rotated rx 180 ry 0 rz 90 deg; joints [76.292, -17.352, 83.721, 0, 23.631, 76.292]
  MoveL 5685 to (27.71, 70.05, -6.88) mm, rotated rx 180 ry 0 rz 90 deg; joints [76.328, -17.352, 83.787, 0, 23.566, 76.328]
  MoveL 5686 to (26.65, 71.15, -7.28) mm, rotated rx 180 ry 0 rz 90 deg; joints [76.355, -17.357, 83.868, 0, 23.488, 76.355]
  MoveL 5687 to (25.38, 71.98, -7.69) mm, rotated rx 180 ry 0 rz 90 deg; joints [76.372, -17.364, 83.961, 0, 23.403, 76.372]
  MoveL 5688 to (23.96, 72.51, -8.09) mm, rotated rx -180 ry 0 rz 90 deg; joints [76.378, -17.372, 84.059, 0, 23.314, 76.378]
  MoveL 5689 to (22.45, 72.69, -8.5) mm, rotated rx 180 ry 0 rz 90 deg; joints [76.372, -17.381, 84.156, 0, 23.224, 76.372]
  MoveL 5690 to (12.79, 72.91, -8.5) mm, rotated rx -180 ry 0 rz 90 deg; joints [76.302, -17.56, 84.852, 0, 22.708, 76.302]
  MoveL 5691 to (-23.4, 73.55, -8.5) mm, rotated rx 180 ry 0 rz 90 deg; joints [76.028, -18.193, 87.408, 0, 20.785, 76.028]
  MoveC 5692 to (-25.87, 70.48, -8.5) mm, rotated rx 180 ry 0 rz 90 deg; joints [75.905, -18.221, 87.526, 0, 20.695, 75.905] to (-25.51, 66.57, -8.5) mm, rotated rx 180 ry 0 rz 90 deg; joints [75.777, -18.199, 87.433, 0, 20.766, 75.777]
  MoveL 5693 to (-9.1, 56.08, -8.5) mm, rotated rx 180 ry 0 rz 90 deg; joints [75.567, -17.875, 86.103, 0, 21.773, 75.567]
  MoveC 5694 to (-8.51, 55.73, -8.5) mm, rotated rx 180 ry 0 rz 90 deg; joints [75.561, -17.864, 86.055, 0, 21.809, 75.561] to (-7.9, 55.44, -8.5) mm, rotated rx -180 ry 0 rz 90 deg; joints [75.556, -17.852, 86.007, 0, 21.845, 75.556]
  MoveC 5695 to (-7.22, 55.43, -8.5) mm, rotated rx 180 ry 0 rz 90 deg; joints [75.562, -17.84, 85.959, 0, 21.881, 75.562] to (-6.55, 55.46, -8.5) mm, rotated rx -180 ry 0 rz 90 deg; joints [75.569, -17.828, 85.912, 0, 21.916, 75.569]
  MoveC 5696 to (9.76, 56.66, -8.5) mm, rotated rx -180 ry 0 rz 90 deg; joints [75.745, -17.542, 84.78, 0, 22.762, 75.745] to (26.06, 58.03, -8.5) mm, rotated rx -180 ry 0 rz 90 deg; joints [75.924, -17.244, 83.636, 0, 23.608, 75.924]
  MoveL 5697 to (29.85, 58.38, -8.5) mm, rotated rx -180 ry 0 rz 90 deg; joints [75.966, -17.173, 83.368, 0, 23.805, 75.966]
  MoveC 5698 to (45.52, 60.04, -8.5) mm, rotated rx -180 ry 0 rz 90 deg; joints [76.145, -16.875, 82.257, 0, 24.618, 76.145] to (61.12, 62.18, -8.5) mm, rotated rx 180 ry 0 rz 90 deg; joints [76.336, -16.568, 81.143, 0, 25.425, 76.336]
  MoveL 5699 to (66.81, 63.13, -8.5) mm, rotated rx 180 ry 0 rz 90 deg; joints [76.41, -16.454, 80.736, 0, 25.718, 76.41]
  MoveL 5700 to (67.79, 63.33, -8.5) mm, rotated rx 180 ry 0 rz 90 deg; joints [76.424, -16.435, 80.667, 0, 25.768, 76.424]
  MoveC 5701 to (69.11, 64.13, -8.5) mm, rotated rx 180 ry 0 rz 90 deg; joints [76.459, -16.411, 80.582, 0, 25.828, 76.459] to (69.61, 65.59, -8.5) mm, rotated rx 180 ry 0 rz 90 deg; joints [76.51, -16.408, 80.571, 0, 25.836, 76.51]
  MoveL 5702 to (69.55, 68.7, -8.5) mm, rotated rx -180 ry 0 rz 90 deg; joints [76.608, -16.425, 80.632, 0, 25.793, 76.608]
  MoveC 5703 to (69.04, 69.59, -8.5) mm, rotated rx -180 ry 0 rz 90 deg; joints [76.633, -16.44, 80.685, 0, 25.755, 76.633] to (68.23, 70.2, -8.5) mm, rotated rx -180 ry 0 rz 90 deg; joints [76.646, -16.46, 80.757, 0, 25.703, 76.646]
  MoveL 5704 to (67.76, 70.29, -8.5) mm, rotated rx 180 ry 0 rz 90 deg; joints [76.645, -16.47, 80.794, 0, 25.677, 76.645]
  MoveL 5705 to (60.14, 70.87, -8.5) mm, rotated rx 180 ry 0 rz 90 deg; joints [76.606, -16.631, 81.371, 0, 25.26, 76.606]
  MoveC 5706 to (42.21, 72, -8.5) mm, rotated rx 180 ry 0 rz 90 deg; joints [76.504, -16.998, 82.712, 0, 24.286, 76.504] to (24.25, 72.65, -8.5) mm, rotated rx 180 ry 0 rz 90 deg; joints [76.385, -17.347, 84.026, 0, 23.32, 76.385]
  MoveL 5707 to (22.45, 72.69, -8.5) mm, rotated rx 180 ry 0 rz 90 deg; joints [76.372, -17.381, 84.156, 0, 23.224, 76.372]
  MoveL 5708 to (22.28, 65.14, -8.5) mm, rotated rx 180 ry 0 rz 90 deg; joints [76.124, -17.349, 84.036, 0, 23.313, 76.124]
  MoveL 5709 to (21.03, 65.17, -8.5) mm, rotated rx -180 ry 0 rz 90 deg; joints [76.115, -17.373, 84.127, 0, 23.246, 76.115]
  MoveL 5710 to (21.03, 65.17, -5.5) mm, rotated rx -180 ry 0 rz 90 deg; joints [76.115, -17.526, 84.228, 0, 23.298, 76.115]
  Establecer velocidad (1000.0 mm/s)
  MoveL 5711 to (21.03, 65.17, 10) mm, rotated rx 180 ry 0 rz 90 deg; joints [76.115, -18.318, 84.746, 0, 23.571, 76.115]
  Establecer velocidad (66.7 mm/s)
  MoveL 5712 to (28.87, 64.04, 10) mm, rotated rx 180 ry 0 rz 90 deg; joints [76.142, -18.162, 84.161, 0, 24.001, 76.142]
  MoveL 5713 to (28.87, 64.04, -5.5) mm, rotated rx -180 ry 0 rz 90 deg; joints [76.142, -17.372, 83.643, 0, 23.73, 76.142]
  MoveL 5714 to (29.1, 65.54, -5.91) mm, rotated rx 180 ry 0 rz 90 deg; joints [76.192, -17.354, 83.639, 0, 23.715, 76.192]
  MoveL 5715 to (28.95, 67.05, -6.31) mm, rotated rx -180 ry 0 rz 90 deg; joints [76.24, -17.343, 83.663, 0, 23.68, 76.24]
  MoveL 5716 to (28.48, 68.49, -6.72) mm, rotated rx -180 ry 0 rz 90 deg; joints [76.283, -17.338, 83.709, 0, 23.629, 76.283]
  MoveL 5717 to (27.7, 69.79, -7.12) mm, rotated rx -180 ry 0 rz 90 deg; joints [76.319, -17.339, 83.775, 0, 23.564, 76.319]
  MoveL 5718 to (26.64, 70.89, -7.53) mm, rotated rx -180 ry 0 rz 90 deg; joints [76.347, -17.343, 83.856, 0, 23.487, 76.347]
  MoveL 5719 to (25.37, 71.73, -7.94) mm, rotated rx -180 ry 0 rz 90 deg; joints [76.364, -17.35, 83.948, 0, 23.402, 76.364]
  MoveL 5720 to (23.95, 72.27, -8.34) mm, rotated rx 180 ry 0 rz 90 deg; joints [76.37, -17.359, 84.046, 0, 23.312, 76.37]
  MoveL 5721 to (22.45, 72.44, -8.75) mm, rotated rx 180 ry 0 rz 90 deg; joints [76.364, -17.367, 84.144, 0, 23.223, 76.364]
  MoveC 5722 to (-0.18, 72.95, -8.75) mm, rotated rx -180 ry 0 rz 90 deg; joints [76.199, -17.781, 85.765, 0, 22.015, 76.199] to (-22.82, 73.33, -8.75) mm, rotated rx -180 ry 0 rz 90 deg; joints [76.026, -18.169, 87.355, 0, 20.814, 76.026]
  MoveC 5723 to (-25.23, 70.3, -8.75) mm, rotated rx -180 ry 0 rz 90 deg; joints [75.904, -18.197, 87.47, 0, 20.727, 75.904] to (-24.87, 66.44, -8.75) mm, rotated rx 180 ry 0 rz 90 deg; joints [75.778, -18.175, 87.378, 0, 20.797, 75.778]
  MoveL 5724 to (-8.82, 56.16, -8.75) mm, rotated rx 180 ry 0 rz 90 deg; joints [75.572, -17.858, 86.076, 0, 21.782, 75.572]
  MoveC 5725 to (-8.27, 55.84, -8.75) mm, rotated rx 180 ry 0 rz 90 deg; joints [75.566, -17.847, 86.031, 0, 21.816, 75.566] to (-7.69, 55.57, -8.75) mm, rotated rx 180 ry 0 rz 90 deg; joints [75.563, -17.836, 85.986, 0, 21.85, 75.563]
  MoveC 5726 to (-6.45, 55.61, -8.75) mm, rotated rx 180 ry 0 rz 90 deg; joints [75.574, -17.814, 85.899, 0, 21.915, 75.574] to (-5.21, 55.68, -8.75) mm, rotated rx 180 ry 0 rz 90 deg; joints [75.587, -17.793, 85.814, 0, 21.979, 75.587]
  MoveL 5727 to (-4.26, 55.77, -8.75) mm, rotated rx 180 ry 0 rz 90 deg; joints [75.598, -17.776, 85.749, 0, 22.028, 75.598]
  MoveC 5728 to (11.95, 57, -8.75) mm, rotated rx 180 ry 0 rz 90 deg; joints [75.774, -17.49, 84.621, 0, 22.869, 75.774] to (28.16, 58.41, -8.75) mm, rotated rx 180 ry 0 rz 90 deg; joints [75.953, -17.193, 83.483, 0, 23.71, 75.953]
  MoveC 5729 to (43.72, 60.08, -8.75) mm, rotated rx -180 ry 0 rz 90 deg; joints [76.132, -16.898, 82.381, 0, 24.517, 76.132] to (59.23, 62.2, -8.75) mm, rotated rx 180 ry 0 rz 90 deg; joints [76.322, -16.594, 81.276, 0, 25.319, 76.322]
  MoveL 5730 to (66.81, 63.51, -8.75) mm, rotated rx 180 ry 0 rz 90 deg; joints [76.422, -16.443, 80.735, 0, 25.709, 76.422]
  MoveL 5731 to (67.64, 63.68, -8.75) mm, rotated rx 180 ry 0 rz 90 deg; joints [76.434, -16.427, 80.675, 0, 25.751, 76.434]
  MoveC 5732 to (68.72, 64.29, -8.75) mm, rotated rx 180 ry 0 rz 90 deg; joints [76.462, -16.407, 80.606, 0, 25.801, 76.462] to (69.24, 65.41, -8.75) mm, rotated rx -180 ry 0 rz 90 deg; joints [76.501, -16.402, 80.587, 0, 25.815, 76.501]
  MoveC 5733 to (69.32, 66.93, -8.75) mm, rotated rx 180 ry 0 rz 90 deg; joints [76.55, -16.408, 80.608, 0, 25.8, 76.55] to (69.2, 68.44, -8.75) mm, rotated rx -180 ry 0 rz 90 deg; joints [76.597, -16.418, 80.644, 0, 25.774, 76.597]
  MoveC 5734 to (68.65, 69.47, -8.75) mm, rotated rx 180 ry 0 rz 90 deg; joints [76.626, -16.435, 80.704, 0, 25.731, 76.626] to (67.58, 69.96, -8.75) mm, rotated rx 180 ry 0 rz 90 deg; joints [76.633, -16.46, 80.792, 0, 25.667, 76.633]
  MoveC 5735 to (45.89, 71.53, -8.75) mm, rotated rx -180 ry 0 rz 90 deg; joints [76.518, -16.91, 82.426, 0, 24.485, 76.518] to (24.17, 72.4, -8.75) mm, rotated rx 180 ry 0 rz 90 deg; joints [76.376, -17.334, 84.02, 0, 23.315, 76.376]
  MoveC 5736 to (23.31, 72.42, -8.75) mm, rotated rx -180 ry 0 rz 90 deg; joints [76.37, -17.351, 84.082, 0, 23.269, 76.37] to (22.45, 72.44, -8.75) mm, rotated rx 180 ry 0 rz 90 deg; joints [76.364, -17.367, 84.144, 0, 23.223, 76.364]
  MoveL 5737 to (22.25, 64.89, -8.75) mm, rotated rx -180 ry 0 rz 90 deg; joints [76.116, -17.336, 84.025, 0, 23.311, 76.116]
  MoveL 5738 to (17.23, 65.02, -8.75) mm, rotated rx 180 ry 0 rz 90 deg; joints [76.08, -17.43, 84.387, 0, 23.043, 76.08]
  MoveL 5739 to (17.23, 65.02, -5.75) mm, rotated rx -180 ry 0 rz 90 deg; joints [76.08, -17.584, 84.489, 0, 23.094, 76.08]
  Establecer velocidad (1000.0 mm/s)
  MoveL 5740 to (17.23, 65.02, 10) mm, rotated rx 180 ry 0 rz 90 deg; joints [76.08, -18.389, 85.016, 0, 23.373, 76.08]
  Establecer velocidad (66.7 mm/s)
  MoveL 5741 to (36.05, 19.91, 10) mm, rotated rx -180 ry 0 rz 90 deg; joints [74.781, -17.794, 82.81, 0, 24.984, 74.781]
  MoveL 5742 to (36.05, 19.91, -5.5) mm, rotated rx 180 ry 0 rz 90 deg; joints [74.781, -17.008, 82.291, 0, 24.718, 74.781]
  MoveL 5743 to (36.21, 21.42, -5.91) mm, rotated rx 180 ry 0 rz 90 deg; joints [74.83, -16.992, 82.294, 0, 24.698, 74.83]
  MoveL 5744 to (36.01, 22.93, -6.31) mm, rotated rx 180 ry 0 rz 90 deg; joints [74.877, -16.984, 82.325, 0, 24.659, 74.877]
  MoveL 5745 to (35.48, 24.35, -6.72) mm, rotated rx 180 ry 0 rz 90 deg; joints [74.918, -16.981, 82.378, 0, 24.604, 74.918]
  MoveL 5746 to (34.65, 25.62, -7.12) mm, rotated rx -180 ry 0 rz 90 deg; joints [74.951, -16.984, 82.449, 0, 24.535, 74.951]
  MoveL 5747 to (33.56, 26.68, -7.53) mm, rotated rx -180 ry 0 rz 90 deg; joints [74.976, -16.991, 82.536, 0, 24.455, 74.976]
  MoveL 5748 to (32.26, 27.47, -7.94) mm, rotated rx -180 ry 0 rz 90 deg; joints [74.99, -17, 82.632, 0, 24.368, 74.99]
  MoveL 5749 to (30.82, 27.95, -8.34) mm, rotated rx 180 ry 0 rz 90 deg; joints [74.993, -17.01, 82.732, 0, 24.278, 74.993]
  MoveL 5750 to (29.31, 28.07, -8.75) mm, rotated rx -180 ry 0 rz 90 deg; joints [74.984, -17.019, 82.83, 0, 24.189, 74.984]
  MoveC 5751 to (20.58, 27.96, -8.75) mm, rotated rx -180 ry 0 rz 90 deg; joints [74.904, -17.187, 83.459, 0, 23.728, 74.904] to (11.85, 27.82, -8.75) mm, rotated rx 180 ry 0 rz 90 deg; joints [74.823, -17.351, 84.082, 0, 23.269, 74.823]
  MoveC 5752 to (9.01, 26.52, -8.75) mm, rotated rx -180 ry 0 rz 90 deg; joints [74.756, -17.397, 84.26, 0, 23.137, 74.756] to (8.05, 23.55, -8.75) mm, rotated rx 180 ry 0 rz 90 deg; joints [74.651, -17.399, 84.27, 0, 23.13, 74.651]
  MoveL 5753 to (8.14, 23.22, -8.75) mm, rotated rx -180 ry 0 rz 90 deg; joints [74.641, -17.396, 84.257, 0, 23.139, 74.641]
  MoveL 5754 to (12.79, 10.5, -8.75) mm, rotated rx -180 ry 0 rz 90 deg; joints [74.272, -17.243, 83.672, 0, 23.571, 74.272]
  MoveL 5755 to (13.01, 9.95, -8.75) mm, rotated rx 180 ry 0 rz 90 deg; joints [74.256, -17.236, 83.645, 0, 23.591, 74.256]
  MoveC 5756 to (13.33, 9.38, -8.75) mm, rotated rx 180 ry 0 rz 90 deg; joints [74.241, -17.227, 83.611, 0, 23.616, 74.241] to (13.78, 8.9, -8.75) mm, rotated rx -180 ry 0 rz 90 deg; joints [74.23, -17.216, 83.569, 0, 23.647, 74.23]
  MoveL 5757 to (14.69, 8.16, -8.75) mm, rotated rx 180 ry 0 rz 90 deg; joints [74.214, -17.195, 83.489, 0, 23.706, 74.214]
  MoveL 5758 to (27.96, -1.91, -8.75) mm, rotated rx 180 ry 0 rz 90 deg; joints [74.013, -16.883, 82.325, 0, 24.558, 74.013]
  MoveL 5759 to (28.9, -2.56, -8.75) mm, rotated rx 180 ry 0 rz 90 deg; joints [74, -16.86, 82.243, 0, 24.618, 74]
  MoveC 5760 to (31.48, -2.65, -8.75) mm, rotated rx -180 ry 0 rz 90 deg; joints [74.021, -16.809, 82.053, 0, 24.756, 74.021] to (33.64, -1.23, -8.75) mm, rotated rx 180 ry 0 rz 90 deg; joints [74.086, -16.774, 81.926, 0, 24.848, 74.086]
  MoveL 5761 to (48.14, 19.43, -8.75) mm, rotated rx 180 ry 0 rz 90 deg; joints [74.869, -16.597, 81.283, 0, 25.313, 74.869]
  MoveL 5762 to (49.33, 21.15, -8.75) mm, rotated rx -180 ry 0 rz 90 deg; joints [74.934, -16.582, 81.23, 0, 25.352, 74.934]
  MoveC 5763 to (49.86, 22.49, -8.75) mm, rotated rx -180 ry 0 rz 90 deg; joints [74.982, -16.578, 81.217, 0, 25.361, 74.982] to (49.75, 23.93, -8.75) mm, rotated rx 180 ry 0 rz 90 deg; joints [75.026, -16.588, 81.254, 0, 25.335, 75.026]
  MoveC 5764 to (48.79, 26.44, -8.75) mm, rotated rx 180 ry 0 rz 90 deg; joints [75.098, -16.622, 81.374, 0, 25.248, 75.098] to (46.78, 28.22, -8.75) mm, rotated rx -180 ry 0 rz 90 deg; joints [75.138, -16.672, 81.557, 0, 25.115, 75.138]
  MoveC 5765 to (38.04, 28.16, -8.75) mm, rotated rx -180 ry 0 rz 90 deg; joints [75.061, -16.848, 82.196, 0, 24.652, 75.061] to (29.31, 28.07, -8.75) mm, rotated rx -180 ry 0 rz 90 deg; joints [74.984, -17.019, 82.83, 0, 24.189, 74.984]
  MoveL 5766 to (29.4, 20.53, -8.75) mm, rotated rx 180 ry 0 rz 90 deg; joints [74.742, -16.978, 82.676, 0, 24.302, 74.742]
  MoveL 5767 to (29.4, 20.53, -5.75) mm, rotated rx 180 ry 0 rz 90 deg; joints [74.742, -17.13, 82.778, 0, 24.353, 74.742]
  Establecer velocidad (1000.0 mm/s)
  MoveL 5768 to (29.4, 20.53, 10) mm, rotated rx 180 ry 0 rz 90 deg; joints [74.742, -17.93, 83.305, 0, 24.625, 74.742]
  Establecer velocidad (66.7 mm/s)
  MoveL 5769 to (62.25, -31.65, 10) mm, rotated rx 180 ry 0 rz 90 deg; joints [73.393, -16.933, 79.787, 0, 27.146, 73.393]
  MoveL 5770 to (62.25, -31.65, -5.5) mm, rotated rx 180 ry 0 rz 90 deg; joints [73.393, -16.156, 79.265, 0, 26.891, 73.393]
  MoveL 5771 to (63.75, -31.89, -5.91) mm, rotated rx -180 ry 0 rz 90 deg; joints [73.399, -16.101, 79.134, 0, 26.968, 73.399]
  MoveL 5772 to (65.26, -31.76, -6.31) mm, rotated rx 180 ry 0 rz 90 deg; joints [73.417, -16.049, 79.009, 0, 27.04, 73.417]
  MoveL 5773 to (66.71, -31.29, -6.72) mm, rotated rx 180 ry 0 rz 90 deg; joints [73.445, -16, 78.897, 0, 27.103, 73.445]
  MoveL 5774 to (68.01, -30.51, -7.12) mm, rotated rx -180 ry 0 rz 90 deg; joints [73.482, -15.956, 78.803, 0, 27.153, 73.482]
  MoveL 5775 to (69.1, -29.44, -7.53) mm, rotated rx 180 ry 0 rz 90 deg; joints [73.524, -15.918, 78.73, 0, 27.188, 73.524]
  MoveL 5776 to (69.92, -28.17, -7.94) mm, rotated rx -180 ry 0 rz 90 deg; joints [73.571, -15.888, 78.683, 0, 27.205, 73.571]
  MoveL 5777 to (70.43, -26.73, -8.34) mm, rotated rx 180 ry 0 rz 90 deg; joints [73.62, -15.866, 78.662, 0, 27.204, 73.62]
  MoveL 5778 to (70.57, -25.22, -8.75) mm, rotated rx -180 ry 0 rz 90 deg; joints [73.668, -15.852, 78.671, 0, 27.181, 73.668]
  MoveL 5779 to (70.57, -18.14, -8.75) mm, rotated rx 180 ry 0 rz 90 deg; joints [73.888, -15.897, 78.827, 0, 27.071, 73.888]
  MoveC 5780 to (69.07, -15.8, -8.75) mm, rotated rx -180 ry 0 rz 90 deg; joints [73.947, -15.945, 78.99, 0, 26.955, 73.947] to (66.81, -14.2, -8.75) mm, rotated rx 180 ry 0 rz 90 deg; joints [73.977, -16.004, 79.195, 0, 26.809, 73.977]
  MoveL 5781 to (66.01, -13.93, -8.75) mm, rotated rx 180 ry 0 rz 90 deg; joints [73.978, -16.024, 79.261, 0, 26.762, 73.978]
  MoveC 5782 to (65.05, -13.74, -8.75) mm, rotated rx 180 ry 0 rz 90 deg; joints [73.975, -16.046, 79.337, 0, 26.708, 73.975] to (64.07, -13.83, -8.75) mm, rotated rx 180 ry 0 rz 90 deg; joints [73.964, -16.066, 79.409, 0, 26.657, 73.964]
  MoveL 5783 to (56.62, -23.92, -8.75) mm, rotated rx 180 ry 0 rz 90 deg; joints [73.581, -16.163, 79.746, 0, 26.417, 73.581]
  MoveC 5784 to (55.99, -26, -8.75) mm, rotated rx -180 ry 0 rz 90 deg; joints [73.511, -16.163, 79.748, 0, 26.416, 73.511] to (56.81, -28, -8.75) mm, rotated rx 180 ry 0 rz 90 deg; joints [73.456, -16.133, 79.642, 0, 26.491, 73.456]
  MoveL 5785 to (64.46, -36.48, -8.75) mm, rotated rx 180 ry 0 rz 90 deg; joints [73.264, -15.913, 78.879, 0, 27.033, 73.264]
  MoveC 5786 to (66.75, -36.25, -8.75) mm, rotated rx -180 ry 0 rz 90 deg; joints [73.292, -15.864, 78.712, 0, 27.152, 73.292] to (68.7, -35.04, -8.75) mm, rotated rx 180 ry 0 rz 90 deg; joints [73.348, -15.829, 78.592, 0, 27.237, 73.348]
  MoveL 5787 to (69.15, -34.59, -8.75) mm, rotated rx 180 ry 0 rz 90 deg; joints [73.366, -15.822, 78.569, 0, 27.253, 73.366]
  MoveC 5788 to (69.97, -33.52, -8.75) mm, rotated rx 180 ry 0 rz 90 deg; joints [73.406, -15.811, 78.531, 0, 27.28, 73.406] to (70.56, -32.31, -8.75) mm, rotated rx 180 ry 0 rz 90 deg; joints [73.449, -15.806, 78.513, 0, 27.293, 73.449]
  MoveL 5789 to (70.57, -31.75, -8.75) mm, rotated rx 180 ry 0 rz 90 deg; joints [73.467, -15.81, 78.525, 0, 27.284, 73.467]
  MoveL 5790 to (70.57, -25.22, -8.75) mm, rotated rx -180 ry 0 rz 90 deg; joints [73.668, -15.852, 78.671, 0, 27.181, 73.668]
  MoveL 5791 to (63.02, -25.22, -8.75) mm, rotated rx -180 ry 0 rz 90 deg; joints [73.6, -16.017, 79.239, 0, 26.778, 73.6]
  MoveL 5792 to (63.02, -25.22, -5.75) mm, rotated rx 180 ry 0 rz 90 deg; joints [73.6, -16.168, 79.342, 0, 26.826, 73.6]
  Establecer velocidad (1000.0 mm/s)
  MoveL 5793 to (63.02, -25.22, 10) mm, rotated rx 180 ry 0 rz 90 deg; joints [73.6, -16.958, 79.873, 0, 27.086, 73.6]
  Establecer velocidad (66.7 mm/s)
  MoveL 5794 to (15.91, -64.62, 10) mm, rotated rx 180 ry 0 rz 90 deg; joints [71.913, -17.69, 82.436, 0, 25.254, 71.913]
  MoveL 5795 to (15.91, -64.62, -5.5) mm, rotated rx -180 ry 0 rz 90 deg; joints [71.913, -16.906, 81.917, 0, 24.989, 71.913]
  MoveL 5796 to (15.76, -66.13, -5.91) mm, rotated rx 180 ry 0 rz 90 deg; joints [71.864, -16.878, 81.878, 0, 25, 71.864]
  MoveL 5797 to (15.98, -67.64, -6.31) mm, rotated rx 180 ry 0 rz 90 deg; joints [71.819, -16.844, 81.813, 0, 25.031, 71.819]
  MoveL 5798 to (16.53, -69.05, -6.72) mm, rotated rx -180 ry 0 rz 90 deg; joints [71.781, -16.803, 81.726, 0, 25.077, 71.781]
  MoveL 5799 to (17.37, -70.31, -7.12) mm, rotated rx -180 ry 0 rz 90 deg; joints [71.75, -16.757, 81.621, 0, 25.136, 71.75]
  MoveL 5800 to (18.48, -71.36, -7.53) mm, rotated rx 180 ry 0 rz 90 deg; joints [71.729, -16.707, 81.502, 0, 25.205, 71.729]
  MoveL 5801 to (19.79, -72.13, -7.94) mm, rotated rx 180 ry 0 rz 90 deg; joints [71.718, -16.655, 81.375, 0, 25.281, 71.718]
  MoveL 5802 to (21.23, -72.59, -8.34) mm, rotated rx 180 ry 0 rz 90 deg; joints [71.719, -16.603, 81.245, 0, 25.358, 71.719]
  MoveL 5803 to (22.75, -72.69, -8.75) mm, rotated rx 180 ry 0 rz 90 deg; joints [71.731, -16.551, 81.119, 0, 25.432, 71.731]
  MoveC 5804 to (34.05, -72.39, -8.75) mm, rotated rx 180 ry 0 rz 90 deg; joints [71.856, -16.321, 80.301, 0, 26.02, 71.856] to (45.35, -72.04, -8.75) mm, rotated rx 180 ry 0 rz 90 deg; joints [71.981, -16.085, 79.475, 0, 26.61, 71.981]
  MoveC 5805 to (47.8, -69.05, -8.75) mm, rotated rx 180 ry 0 rz 90 deg; joints [72.098, -16.054, 79.365, 0, 26.688, 72.098] to (47.94, -65.19, -8.75) mm, rotated rx -180 ry 0 rz 90 deg; joints [72.218, -16.077, 79.447, 0, 26.63, 72.218]
  MoveC 5806 to (36.54, -51.56, -8.75) mm, rotated rx 180 ry 0 rz 90 deg; joints [72.529, -16.408, 80.609, 0, 25.799, 72.529] to (25.07, -37.98, -8.75) mm, rotated rx 180 ry 0 rz 90 deg; joints [72.842, -16.727, 81.755, 0, 24.972, 72.842]
  MoveC 5807 to (24.53, -37.41, -8.75) mm, rotated rx 180 ry 0 rz 90 deg; joints [72.855, -16.741, 81.807, 0, 24.934, 72.855] to (23.94, -36.88, -8.75) mm, rotated rx -180 ry 0 rz 90 deg; joints [72.866, -16.756, 81.862, 0, 24.894, 72.866]
  MoveL 5808 to (12.79, -27.86, -8.75) mm, rotated rx 180 ry 0 rz 90 deg; joints [73.044, -17.029, 82.866, 0, 24.163, 73.044]
  MoveC 5809 to (10.57, -27.28, -8.75) mm, rotated rx -180 ry 0 rz 90 deg; joints [73.041, -17.075, 83.038, 0, 24.037, 73.041] to (8.37, -27.96, -8.75) mm, rotated rx 180 ry 0 rz 90 deg; joints [72.998, -17.113, 83.18, 0, 23.933, 72.998]
  MoveL 5810 to (8.17, -28.08, -8.75) mm, rotated rx -180 ry 0 rz 90 deg; joints [72.992, -17.116, 83.192, 0, 23.924, 72.992]
  MoveC 5811 to (7.49, -28.72, -8.75) mm, rotated rx 180 ry 0 rz 90 deg; joints [72.965, -17.125, 83.227, 0, 23.898, 72.965] to (7.08, -29.56, -8.75) mm, rotated rx 180 ry 0 rz 90 deg; joints [72.934, -17.128, 83.237, 0, 23.891, 72.934]
  MoveL 5812 to (-3.44, -68.7, -8.75) mm, rotated rx -180 ry 0 rz 90 deg; joints [71.584, -17.09, 83.095, 0, 23.995, 71.584]
  MoveC 5813 to (-3.38, -70.55, -8.75) mm, rotated rx -180 ry 0 rz 90 deg; joints [71.526, -17.077, 83.047, 0, 24.03, 71.526] to (-2.37, -72.1, -8.75) mm, rotated rx 180 ry 0 rz 90 deg; joints [71.488, -17.048, 82.938, 0, 24.11, 71.488]
  MoveC 5814 to (-1.23, -72.89, -8.75) mm, rotated rx -180 ry 0 rz 90 deg; joints [71.475, -17.021, 82.838, 0, 24.183, 71.475] to (0.13, -73.15, -8.75) mm, rotated rx -180 ry 0 rz 90 deg; joints [71.481, -16.994, 82.735, 0, 24.259, 71.481]
  MoveC 5815 to (11.44, -72.95, -8.75) mm, rotated rx 180 ry 0 rz 90 deg; joints [71.606, -16.775, 81.93, 0, 24.845, 71.606] to (22.75, -72.69, -8.75) mm, rotated rx 180 ry 0 rz 90 deg; joints [71.731, -16.551, 81.119, 0, 25.432, 71.731]
  MoveL 5816 to (22.56, -65.15, -8.75) mm, rotated rx -180 ry 0 rz 90 deg; joints [71.965, -16.605, 81.312, 0, 25.293, 71.965]
  MoveL 5817 to (22.56, -65.15, -5.75) mm, rotated rx -180 ry 0 rz 90 deg; joints [71.965, -16.756, 81.414, 0, 25.342, 71.965]
  Establecer velocidad (1000.0 mm/s)
  MoveL 5818 to (22.56, -65.15, 10) mm, rotated rx 180 ry 0 rz 90 deg; joints [71.965, -17.552, 81.943, 0, 25.609, 71.965]
  Establecer velocidad (66.7 mm/s)
  MoveL 5819 to (-36.11, -51.64, 10) mm, rotated rx 180 ry 0 rz 90 deg; joints [71.784, -18.748, 86.406, 0, 22.342, 71.784]
  MoveL 5820 to (-36.11, -51.64, -5.5) mm, rotated rx 180 ry 0 rz 90 deg; joints [71.784, -17.951, 85.888, 0, 22.063, 71.784]
  MoveL 5821 to (-34.7, -52.19, -5.91) mm, rotated rx -180 ry 0 rz 90 deg; joints [71.781, -17.903, 85.764, 0, 22.138, 71.781]
  MoveL 5822 to (-33.2, -52.4, -6.31) mm, rotated rx -180 ry 0 rz 90 deg; joints [71.79, -17.854, 85.642, 0, 22.213, 71.79]
  MoveL 5823 to (-31.68, -52.26, -6.72) mm, rotated rx 180 ry 0 rz 90 deg; joints [71.81, -17.808, 85.526, 0, 22.282, 71.81]
  MoveL 5824 to (-30.23, -51.8, -7.12) mm, rotated rx 180 ry 0 rz 90 deg; joints [71.841, -17.764, 85.423, 0, 22.341, 71.841]
  MoveL 5825 to (-28.93, -51.02, -7.53) mm, rotated rx 180 ry 0 rz 90 deg; joints [71.88, -17.725, 85.336, 0, 22.389, 71.88]
  MoveL 5826 to (-27.83, -49.97, -7.94) mm, rotated rx 180 ry 0 rz 90 deg; joints [71.925, -17.691, 85.269, 0, 22.421, 71.925]
  MoveL 5827 to (-26.98, -48.71, -8.34) mm, rotated rx -180 ry 0 rz 90 deg; joints [71.974, -17.662, 85.225, 0, 22.437, 71.974]
  MoveL 5828 to (-26.46, -47.28, -8.75) mm, rotated rx -180 ry 0 rz 90 deg; joints [72.026, -17.64, 85.208, 0, 22.432, 72.026]
  MoveL 5829 to (-20.36, -23.79, -8.75) mm, rotated rx -180 ry 0 rz 90 deg; joints [72.848, -17.664, 85.3, 0, 22.363, 72.848]
  MoveC 5830 to (-20.29, -23.26, -8.75) mm, rotated rx 180 ry 0 rz 90 deg; joints [72.866, -17.665, 85.307, 0, 22.358, 72.866] to (-20.36, -22.74, -8.75) mm, rotated rx 180 ry 0 rz 90 deg; joints [72.882, -17.669, 85.323, 0, 22.346, 72.882]
  MoveC 5831 to (-21.41, -20.87, -8.75) mm, rotated rx 180 ry 0 rz 90 deg; joints [72.932, -17.698, 85.436, 0, 22.262, 72.932] to (-23.22, -19.72, -8.75) mm, rotated rx -180 ry 0 rz 90 deg; joints [72.951, -17.736, 85.587, 0, 22.149, 72.951]
  MoveC 5832 to (-23.71, -19.63, -8.75) mm, rotated rx -180 ry 0 rz 90 deg; joints [72.949, -17.745, 85.624, 0, 22.122, 72.949] to (-24.21, -19.67, -8.75) mm, rotated rx -180 ry 0 rz 90 deg; joints [72.943, -17.754, 85.658, 0, 22.096, 72.943]
  MoveC 5833 to (-47.88, -24.65, -8.75) mm, rotated rx -180 ry 0 rz 90 deg; joints [72.54, -18.128, 87.183, 0, 20.945, 72.54] to (-71.55, -29.66, -8.75) mm, rotated rx -180 ry 0 rz 90 deg; joints [72.126, -18.479, 88.676, 0, 19.803, 72.126]
  MoveC 5834 to (-73.37, -30.72, -8.75) mm, rotated rx 180 ry 0 rz 90 deg; joints [72.071, -18.502, 88.776, 0, 19.726, 72.071] to (-74.14, -32.69, -8.75) mm, rotated rx -180 ry 0 rz 90 deg; joints [71.997, -18.503, 88.784, 0, 19.719, 71.997]
  MoveL 5835 to (-74.15, -33.64, -8.75) mm, rotated rx 180 ry 0 rz 90 deg; joints [71.965, -18.499, 88.764, 0, 19.735, 71.965]
  MoveL 5836 to (-74.15, -69.65, -8.75) mm, rotated rx 180 ry 0 rz 90 deg; joints [70.778, -18.31, 87.951, 0, 20.36, 70.778]
  MoveL 5837 to (-74.14, -70.4, -8.75) mm, rotated rx 180 ry 0 rz 90 deg; joints [70.754, -18.306, 87.932, 0, 20.374, 70.754]
  MoveC 5838 to (-73.16, -72.65, -8.75) mm, rotated rx -180 ry 0 rz 90 deg; joints [70.691, -18.278, 87.814, 0, 20.464, 70.691] to (-70.87, -73.56, -8.75) mm, rotated rx 180 ry 0 rz 90 deg; joints [70.688, -18.237, 87.639, 0, 20.598, 70.688]
  MoveL 5839 to (-36.48, -73.25, -8.75) mm, rotated rx -180 ry 0 rz 90 deg; joints [71.083, -17.664, 85.302, 0, 22.362, 71.083]
  MoveL 5840 to (-35.67, -73.23, -8.75) mm, rotated rx 180 ry 0 rz 90 deg; joints [71.093, -17.65, 85.246, 0, 22.404, 71.093]
  MoveC 5841 to (-33.71, -72.53, -8.75) mm, rotated rx 180 ry 0 rz 90 deg; joints [71.137, -17.62, 85.127, 0, 22.492, 71.137] to (-32.58, -70.78, -8.75) mm, rotated rx 180 ry 0 rz 90 deg; joints [71.205, -17.61, 85.09, 0, 22.52, 71.205]
  MoveL 5842 to (-26.46, -47.28, -8.75) mm, rotated rx -180 ry 0 rz 90 deg; joints [72.026, -17.64, 85.208, 0, 22.432, 72.026]
  MoveL 5843 to (-33.77, -45.38, -8.75) mm, rotated rx -180 ry 0 rz 90 deg; joints [72.011, -17.779, 85.757, 0, 22.021, 72.011]
  MoveL 5844 to (-33.77, -45.38, -5.75) mm, rotated rx 180 ry 0 rz 90 deg; joints [72.011, -17.933, 85.859, 0, 22.074, 72.011]
  Establecer velocidad (1000.0 mm/s)
  MoveL 5845 to (-33.77, -45.38, 10) mm, rotated rx 180 ry 0 rz 90 deg; joints [72.011, -18.743, 86.385, 0, 22.358, 72.011]
  Establecer velocidad (66.7 mm/s)
  MoveL 5846 to (-65.91, 36.27, 10) mm, rotated rx -180 ry 0 rz 90 deg; joints [74.394, -19.675, 90.258, 0, 19.418, 74.394]
  MoveL 5847 to (-65.91, 36.27, -5.5) mm, rotated rx -180 ry 0 rz 90 deg; joints [74.394, -18.864, 89.74, 0, 19.125, 74.394]
  MoveL 5848 to (-67.42, 36.46, -5.91) mm, rotated rx -180 ry 0 rz 90 deg; joints [74.386, -18.866, 89.831, 0, 19.036, 74.386]
  MoveL 5849 to (-68.93, 36.27, -6.31) mm, rotated rx -180 ry 0 rz 90 deg; joints [74.366, -18.867, 89.915, 0, 18.952, 74.366]
  MoveL 5850 to (-70.36, 35.76, -6.72) mm, rotated rx 180 ry 0 rz 90 deg; joints [74.335, -18.864, 89.987, 0, 18.877, 74.335]
  MoveL 5851 to (-71.64, 34.95, -7.12) mm, rotated rx 180 ry 0 rz 90 deg; joints [74.295, -18.859, 90.044, 0, 18.815, 74.295]
  MoveL 5852 to (-72.71, 33.87, -7.53) mm, rotated rx 180 ry 0 rz 90 deg; joints [74.248, -18.848, 90.081, 0, 18.767, 74.248]
  MoveL 5853 to (-73.52, 32.58, -7.94) mm, rotated rx 180 ry 0 rz 90 deg; joints [74.196, -18.834, 90.097, 0, 18.737, 74.196]
  MoveL 5854 to (-74.01, 31.14, -8.34) mm, rotated rx -180 ry 0 rz 90 deg; joints [74.143, -18.814, 90.089, 0, 18.725, 74.143]
  MoveL 5855 to (-74.15, 29.63, -8.75) mm, rotated rx -180 ry 0 rz 90 deg; joints [74.09, -18.788, 90.056, 0, 18.732, 74.09]
  MoveL 5856 to (-74.15, 2.37, -8.75) mm, rotated rx 180 ry 0 rz 90 deg; joints [73.169, -18.67, 89.521, 0, 19.149, 73.169]
  MoveL 5857 to (-74.14, 1.42, -8.75) mm, rotated rx 180 ry 0 rz 90 deg; joints [73.137, -18.665, 89.501, 0, 19.164, 73.137]
  MoveC 5858 to (-73.07, -0.98, -8.75) mm, rotated rx 180 ry 0 rz 90 deg; joints [73.067, -18.638, 89.38, 0, 19.258, 73.067] to (-70.6, -1.88, -8.75) mm, rotated rx 180 ry 0 rz 90 deg; joints [73.062, -18.597, 89.197, 0, 19.401, 73.062]
  MoveL 5859 to (-69.65, -1.69, -8.75) mm, rotated rx 180 ry 0 rz 90 deg; joints [73.078, -18.584, 89.137, 0, 19.447, 73.078]
  MoveL 5860 to (-62.07, 0.06, -8.75) mm, rotated rx 180 ry 0 rz 90 deg; joints [73.214, -18.476, 88.662, 0, 19.813, 73.214]
  MoveL 5861 to (-23.46, 9, -8.75) mm, rotated rx 180 ry 0 rz 90 deg; joints [73.887, -17.888, 86.199, 0, 21.689, 73.887]
  MoveL 5862 to (-22.27, 9.28, -8.75) mm, rotated rx -180 ry 0 rz 90 deg; joints [73.908, -17.869, 86.122, 0, 21.747, 73.908]
  MoveL 5863 to (-21.8, 9.4, -8.75) mm, rotated rx 180 ry 0 rz 90 deg; joints [73.916, -17.862, 86.091, 0, 21.77, 73.916]
  MoveC 5864 to (-19.86, 10.88, -8.75) mm, rotated rx 180 ry 0 rz 90 deg; joints [73.983, -17.836, 85.986, 0, 21.849, 73.983] to (-19.34, 13.27, -8.75) mm, rotated rx 180 ry 0 rz 90 deg; joints [74.066, -17.838, 85.997, 0, 21.841, 74.066]
  MoveL 5865 to (-19.48, 13.74, -8.75) mm, rotated rx 180 ry 0 rz 90 deg; joints [74.08, -17.843, 86.017, 0, 21.827, 74.08]
  MoveL 5866 to (-21.32, 18.92, -8.75) mm, rotated rx 180 ry 0 rz 90 deg; joints [74.233, -17.9, 86.248, 0, 21.653, 74.233]
  MoveL 5867 to (-25.85, 31.61, -8.75) mm, rotated rx -180 ry 0 rz 90 deg; joints [74.61, -18.038, 86.808, 0, 21.229, 74.61]
  MoveC 5868 to (-26.2, 32.37, -8.75) mm, rotated rx 180 ry 0 rz 90 deg; joints [74.632, -18.047, 86.847, 0, 21.2, 74.632] to (-26.68, 33.06, -8.75) mm, rotated rx 180 ry 0 rz 90 deg; joints [74.651, -18.058, 86.893, 0, 21.165, 74.651]
  MoveC 5869 to (-27.14, 33.42, -8.75) mm, rotated rx 180 ry 0 rz 90 deg; joints [74.658, -18.067, 86.931, 0, 21.136, 74.658] to (-27.61, 33.75, -8.75) mm, rotated rx 180 ry 0 rz 90 deg; joints [74.665, -18.077, 86.97, 0, 21.106, 74.665]
  MoveL 5870 to (-36.48, 39.47, -8.75) mm, rotated rx -180 ry 0 rz 90 deg; joints [74.775, -18.249, 87.69, 0, 20.559, 74.775]
  MoveL 5871 to (-66.81, 58.94, -8.75) mm, rotated rx -180 ry 0 rz 90 deg; joints [75.157, -18.798, 90.104, 0, 18.695, 75.157]
  MoveL 5872 to (-69.52, 60.65, -8.75) mm, rotated rx -180 ry 0 rz 90 deg; joints [75.191, -18.845, 90.316, 0, 18.529, 75.191]
  MoveC 5873 to (-71.78, 60.58, -8.75) mm, rotated rx -180 ry 0 rz 90 deg; joints [75.168, -18.877, 90.466, 0, 18.411, 75.168] to (-73.59, 59.23, -8.75) mm, rotated rx -180 ry 0 rz 90 deg; joints [75.105, -18.898, 90.563, 0, 18.335, 75.105]
  MoveL 5874 to (-73.87, 58.81, -8.75) mm, rotated rx 180 ry 0 rz 90 deg; joints [75.089, -18.9, 90.574, 0, 18.327, 75.089]
  MoveC 5875 to (-74.08, 58.35, -8.75) mm, rotated rx 180 ry 0 rz 90 deg; joints [75.071, -18.902, 90.58, 0, 18.322, 75.071] to (-74.15, 57.84, -8.75) mm, rotated rx 180 ry 0 rz 90 deg; joints [75.053, -18.901, 90.576, 0, 18.325, 75.053]
  MoveL 5876 to (-74.15, 29.63, -8.75) mm, rotated rx -180 ry 0 rz 90 deg; joints [74.09, -18.788, 90.056, 0, 18.732, 74.09]
  MoveL 5877 to (-66.6, 29.63, -8.75) mm, rotated rx 180 ry 0 rz 90 deg; joints [74.163, -18.676, 89.55, 0, 19.126, 74.163]
  MoveL 5878 to (-66.6, 29.63, -5.75) mm, rotated rx -180 ry 0 rz 90 deg; joints [74.163, -18.833, 89.652, 0, 19.181, 74.163]
  Establecer velocidad (1000.0 mm/s)
  MoveL 5879 to (-66.6, 29.63, 10) mm, rotated rx 180 ry 0 rz 90 deg; joints [74.163, -19.657, 90.178, 0, 19.479, 74.163]
  Establecer velocidad (66.7 mm/s)
  MoveL 5880 to (-65.75, 36.27, 10) mm, rotated rx 180 ry 0 rz 90 deg; joints [74.396, -19.673, 90.246, 0, 19.426, 74.396]
  MoveL 5881 to (-65.75, 36.27, -5.75) mm, rotated rx -180 ry 0 rz 90 deg; joints [74.396, -18.849, 89.72, 0, 19.129, 74.396]
  MoveL 5882 to (-67.25, 36.46, -6.16) mm, rotated rx -180 ry 0 rz 90 deg; joints [74.388, -18.851, 89.811, 0, 19.04, 74.388]
  MoveL 5883 to (-68.76, 36.27, -6.56) mm, rotated rx 180 ry 0 rz 90 deg; joints [74.367, -18.851, 89.895, 0, 18.956, 74.367]
  MoveL 5884 to (-70.19, 35.76, -6.97) mm, rotated rx 180 ry 0 rz 90 deg; joints [74.336, -18.849, 89.967, 0, 18.881, 74.336]
  MoveL 5885 to (-71.48, 34.95, -7.38) mm, rotated rx -180 ry 0 rz 90 deg; joints [74.296, -18.843, 90.024, 0, 18.819, 74.296]
  MoveL 5886 to (-72.54, 33.87, -7.78) mm, rotated rx -180 ry 0 rz 90 deg; joints [74.249, -18.833, 90.062, 0, 18.771, 74.249]
  MoveL 5887 to (-73.35, 32.58, -8.19) mm, rotated rx 180 ry 0 rz 90 deg; joints [74.198, -18.818, 90.077, 0, 18.741, 74.198]
  MoveL 5888 to (-73.85, 31.14, -8.59) mm, rotated rx -180 ry 0 rz 90 deg; joints [74.144, -18.798, 90.07, 0, 18.728, 74.144]
  MoveL 5889 to (-73.99, 29.63, -9) mm, rotated rx 180 ry 0 rz 90 deg; joints [74.092, -18.773, 90.036, 0, 18.736, 74.092]
  MoveL 5890 to (-73.99, 2.37, -9) mm, rotated rx 180 ry 0 rz 90 deg; joints [73.17, -18.654, 89.501, 0, 19.153, 73.17]
  MoveL 5891 to (-73.97, 1.42, -9) mm, rotated rx -180 ry 0 rz 90 deg; joints [73.139, -18.65, 89.481, 0, 19.169, 73.139]
  MoveC 5892 to (-72.91, -0.81, -9) mm, rotated rx -180 ry 0 rz 90 deg; joints [73.074, -18.624, 89.364, 0, 19.259, 73.074] to (-70.6, -1.7, -9) mm, rotated rx 180 ry 0 rz 90 deg; joints [73.068, -18.585, 89.192, 0, 19.393, 73.068]
  MoveL 5893 to (-69.65, -1.53, -9) mm, rotated rx 180 ry 0 rz 90 deg; joints [73.084, -18.571, 89.132, 0, 19.44, 73.084]
